# B&R Automation Studio project Nitto (part 7)

#### SPR_LabelerAut.st - Cam automat configuration for labeling unit
```iecst
(********************************************************************
 * COPYRIGHT -- Bernecker + Rainer
 ********************************************************************
 * Library: UserSpilke
 * File: SPR_LabelerAut.st
 * Author: knausenbergl
 * Created: January 30, 2013
 ********************************************************************
 * Implementation of library UserSpilke
 ********************************************************************)

(*<$Description$> Cam automat configuration for labeling unit </$Description$>*)
FUNCTION_BLOCK SPR_LabelerAut

	//********************	GLOBAL AUTOMAT CONFIGURATION ********************
	AutData.Master				:= Master;
	AutData.MaxMasterVelocity	:= MaxMasterVelocity;
	AutData.SlaveLatchParID		:= ACP10PAR_AUT_SL_S;
	AutData.StartState			:= 0;
	//***********************************************************************

	//********************	STATE 0: INIT ********************
	//state transition
	AutData.State[0].Event[0].Type		:= ncST_END;
	AutData.State[0].Event[0].Attribute	:= ncAT_ONCE;
	AutData.State[0].Event[0].NextState	:= 1;
	//********************************************************

	//********************	STATE 1: ALIGN MIDDLE OF CAM WITH REG MARK	********************
	//compensation
	AutData.State[1].CompMode	:= ncOFF;

	//cam profile
	AutData.State[1].CamProfileIndex	:= 16#FFFF;
//	AutData.State[1].MasterFactor		:= REAL_TO_UDINT(fmod( (LabelPeriod / 2.0 - DistanceToLabelSensor) , LabelPeriod) + 2.0 * LabelPeriod);
	AutData.State[1].MasterFactor		:= REAL_TO_UDINT(fmod( ABS(LabelPeriod / 2.0 - DistanceToLabelSensor) , LabelPeriod) + 2.0 * LabelPeriod);

	AutData.State[1].SlaveFactor		:= UDINT_TO_DINT(AutData.State[1].MasterFactor);

	//state transition
	AutData.State[1].Event[0].Type		:= ncST_END;
	AutData.State[1].Event[0].Attribute	:= ncAT_ONCE;
	AutData.State[1].Event[0].NextState	:= 2;
	//**************************************************************************************

	//********************	STATE 2: STANDARD CAM WITHOUT CORRECTION ********************
	//compensation
	AutData.State[2].CompMode			:= ncOFF;

	//cam profile
	AutData.State[2].CamProfileIndex	:= 16#FFFF;
	AutData.State[2].MasterFactor		:= REAL_TO_UDINT(LabelPeriod);
	AutData.State[2].SlaveFactor		:= REAL_TO_DINT(LabelPeriod);

	//state transition
	AutData.State[2].Event[0].Type		:= TriggerEvent;
	AutData.State[2].Event[0].Attribute	:= ncAT_ONCE;
	AutData.State[2].Event[0].NextState	:= 3;
	//************************************************************************

	//********************	STATE 3: LABEL POSITION CORRECTION	********************
	//compensation
	AutData.State[3].CompMode			:= ncSL_LATCHPOS;
	AutData.State[3].SlaveCompDistance	:= LabelPeriod;
	AutData.State[3].MasterCompDistance	:= LabelPeriod;

	//cam profile
	AutData.State[3].CamProfileIndex	:= 16#FFFE;
	AutData.State[3].MasterFactor		:= REAL_TO_UDINT(LabelPeriod);
	AutData.State[3].SlaveFactor		:= REAL_TO_DINT(LabelPeriod);

	//state transition
	AutData.State[3].Event[0].Type		:= TriggerEvent;
	AutData.State[3].Event[0].Attribute	:= ncAT_ONCE;
	AutData.State[3].Event[0].NextState	:= 3;

	AutData.State[3].Event[1].Type		:= ncST_END;
	AutData.State[3].Event[1].Attribute	:= ncAT_ONCE;
	AutData.State[3].Event[1].NextState	:= 4;
	//******************************************************************************

	//********************	STATE 4: POINT-TO-POINT CAM  WITHOUT CORRECTION	********************
	//compensation
	AutData.State[4].CompMode			:= ncWITH_CAM;
	AutData.State[4].SlaveCompDistance	:= LabelPeriod;
	AutData.State[4].MasterCompDistance	:= LabelPeriod;

	//cam profile
	AutData.State[4].CamProfileIndex	:= 16#FFFE;
	AutData.State[4].MasterFactor		:= REAL_TO_UDINT(LabelPeriod);
	AutData.State[4].SlaveFactor		:= REAL_TO_DINT(LabelPeriod);

	//state transition
	AutData.State[4].Event[0].Type		:= TriggerEvent;
	AutData.State[4].Event[0].Attribute	:= ncAT_ONCE;
	AutData.State[4].Event[0].NextState	:= 3;
	//*******************************************************************************************

	//ignore other states
	AutData.State[0].DisableStateInit	:= ncOFF;
	AutData.State[1].DisableStateInit	:= ncOFF;
	AutData.State[2].DisableStateInit	:= ncOFF;
	AutData.State[3].DisableStateInit	:= ncOFF;
	AutData.State[4].DisableStateInit	:= ncOFF;
	AutData.State[5].DisableStateInit	:= ncON;
	AutData.State[6].DisableStateInit	:= ncON;
	AutData.State[7].DisableStateInit	:= ncON;
	AutData.State[8].DisableStateInit	:= ncON;
	AutData.State[9].DisableStateInit	:= ncON;
	AutData.State[10].DisableStateInit	:= ncON;
	AutData.State[11].DisableStateInit	:= ncON;
	AutData.State[12].DisableStateInit	:= ncON;
	AutData.State[13].DisableStateInit	:= ncON;
	AutData.State[14].DisableStateInit	:= ncON;

	adrAutData	:= ADR(AutData);

END_FUNCTION_BLOCK
```

#### SPR_LabelerAutVax.st - Cam automat configuration for an "ideal" labeler (no label position correction)
```iecst
(********************************************************************
 * COPYRIGHT -- Bernecker + Rainer
 ********************************************************************
 * Library: UserSpilke
 * File: SPR_LabelerAutVax.st
 * Author: knausenbergl
 * Created: February 02, 2013
 ********************************************************************
 * Implementation of library UserSpilke
 ********************************************************************)

(*<$Description$> Cam automat configuration for an "ideal" labeler (no label position correction) </$Description$>*)
FUNCTION_BLOCK SPR_LabelerAutVax

	//the sum of acceleration distance, cam length and deceleration distance equals 1 label period
	IF ( (AccelerationBias >= 0.1) AND (AccelerationBias <= 10.0) ) THEN
		AccelerationDistance	:= (LabelPeriod - CamLength) * AccelerationBias / (AccelerationBias + 1.0);
	ELSE
		AccelerationDistance	:= (LabelPeriod - CamLength) / 2.0;	//default value
	END_IF;
	DecelerationDistance	:= LabelPeriod - CamLength - AccelerationDistance;

	//********************	GLOBAL AUTOMAT CONFIGURATION ********************
	AutData.Master				:= Master;
	AutData.MaxMasterVelocity	:= MaxMasterVelocity;
	AutData.StartState			:= 0;
	//***********************************************************************

	//********************	STATE 0: INIT ********************
	//state transition
	AutData.State[0].Event[0].Type		:= ncST_END;
	AutData.State[0].Event[0].Attribute	:= ncAT_ONCE;
	AutData.State[0].Event[0].NextState	:= 1;
	//********************************************************

	//********************	STATE 1: STANDSTILL, WAIT FOR TRIGGER EVENT	********************
	//compensation
	AutData.State[1].CompMode	:= ncOFF;

	//cam profile
	AutData.State[1].CamProfileIndex	:= 16#FFFF;
	AutData.State[1].MasterFactor		:= REAL_TO_UDINT(ProductLengthMaster);
	AutData.State[1].SlaveFactor		:= REAL_TO_DINT(LabelPeriod);

	//state transition
	AutData.State[1].Event[0].Type		:= ncSIGNAL1;
	AutData.State[1].Event[0].Attribute	:= ncAT_ONCE;
	AutData.State[1].Event[0].NextState	:= 2;

	AutData.State[1].Event[1].Type		:= TriggerEvent;	//reg mark found
	AutData.State[1].Event[1].Attribute	:= ncAT_ONCE;
	AutData.State[1].Event[1].NextState	:= 2;
	//**************************************************************************************

	//********************	STATE 2: DISPENSE FIRST LABEL ********************
	//compensation
//	AutData.State[2].CompMode			:= ncMA_LATCHPOS;
//	AutData.State[2].SlaveCompDistance	:= AccelerationDistance + 0.5 * CamLength;
//	AutData.State[2].MasterCompDistance	:= fmod( (DistanceToRmSensor - RegMarkPosition), ProductLengthMaster) + ProductLengthMaster;	//distance from sensor to middle of label

	// okrebs 12.09.13
	AutData.State[2].CompMode			:= ncMA_LATCHPOS;
	AutData.State[2].SlaveCompDistance	:= AccelerationDistance + 0.5 * LabelPeriod;
	AutData.State[2].MasterCompDistance	:= fmod( (DistanceToRmSensor - RegMarkPosition), ProductLengthMaster) + ProductLengthMaster;	//distance from sensor to middle of label

	//	//cam profile
    AutData.State[2].CamProfileIndex	:= 16#FFFF;
//	AutData.State[2].MasterFactor		:= REAL_TO_UDINT(CamLength);
//	AutData.State[2].SlaveFactor		:= REAL_TO_DINT(CamLength);

	IF (ProductLengthMaster > 0.0) THEN
		AutData.State[2].SlaveFactor		:= REAL_TO_DINT(LabelPeriod * LabelPeriod / ProductLengthMaster);
		AutData.State[2].MasterFactor		:= REAL_TO_UDINT(LabelPeriod);
	ELSE
		// Invalid parameters, use fix values
		AutData.State[2].MasterFactor		:= REAL_TO_UDINT(CamLength);
		AutData.State[2].SlaveFactor		:= REAL_TO_DINT(CamLength);
	END_IF

	//state transition
	AutData.State[2].Event[0].Type		:= ncST_END;
	AutData.State[2].Event[0].Attribute	:= ncAT_ONCE;
	AutData.State[2].Event[0].NextState	:= 3;

	AutData.State[2].Event[1].Type		:= ncSIGNAL2;	//stop labelling
	AutData.State[2].Event[1].Attribute	:= ncST_END;
	AutData.State[2].Event[1].NextState	:= 5;
	//************************************************************************

	//********************	STATE 3: CYCLIC LABELING WITHOUT CORRECTION	********************
	//compensation
	// AutData.State[3].CompMode			:= ncWITH_CAM;

	// okrebs 12.09.13
	 AutData.State[3].CompMode			:= ncOFF;

	AutData.State[3].SlaveCompDistance	:= LabelPeriod;			//label period on slave
	AutData.State[3].MasterCompDistance	:= ProductLengthMaster;	//distance label to label on master

//	//cam profile
//	AutData.State[3].CamProfileIndex	:= 16#FFFF;
//	AutData.State[3].MasterFactor		:= REAL_TO_UDINT(CamLength);
//	AutData.State[3].SlaveFactor		:= REAL_TO_DINT(CamLength);

	// okrebs / schoenefeldr 13.09.13
	AutData.State[3].CamProfileIndex	:= 16#FFFF;
	// Original:          SlaveFactor         Label period
	//            Gear = -------------- = -----------------------
	//                    MasterFactor      ProductLengthMaster
	// Use label period for the master cam length as it will be significantly
	// shorter than ProductLengthMaster -> so there is enough master distance
	// left for compensation:
	//           Label period                  Label period * (Label period / ProductLengthMaster)
	//   Gear = -----------------------  =   -------------------------
	//           ProductLengthMaster           Label period
	IF (ProductLengthMaster > 0.0) THEN
		AutData.State[3].SlaveFactor		:= REAL_TO_DINT(LabelPeriod * LabelPeriod / ProductLengthMaster);
		AutData.State[3].MasterFactor		:= REAL_TO_UDINT(LabelPeriod);
	ELSE
		// Invalid parameters, use fix values
		AutData.State[3].MasterFactor		:= REAL_TO_UDINT(CamLength);
		AutData.State[3].SlaveFactor		:= REAL_TO_DINT(CamLength);
	END_IF

	//state transition
	AutData.State[3].Event[0].Type		:= TriggerEvent;
	AutData.State[3].Event[0].Attribute	:= ncST_END;
	AutData.State[3].Event[0].NextState	:= 4;

	AutData.State[3].Event[1].Type		:= ncSIGNAL2;	//stop labelling
	AutData.State[3].Event[1].Attribute	:= ncST_END;
	AutData.State[3].Event[1].NextState	:= 5;

	//***************************************************************************************

	//********************	STATE 4: CYCLIC LABELING WITH CORRECTION	********************
	//compensation
	AutData.State[4].CompMode			:= ncMA_LATCHPOS;
	AutData.State[4].SlaveCompDistance	:= LabelPeriod;								//label period on slave
	AutData.State[4].MasterCompDistance	:= fmod( (DistanceToRmSensor - RegMarkPosition), ProductLengthMaster) + ProductLengthMaster;	//distance from sensor to middle of label

//	//cam profile
//	AutData.State[4].CamProfileIndex	:= 16#FFFF;
//	AutData.State[4].MasterFactor		:= REAL_TO_UDINT(CamLength);
//	AutData.State[4].SlaveFactor		:= REAL_TO_DINT(CamLength);

	// okrebs 12.09.13
	AutData.State[4].CamProfileIndex	:= 16#FFFF;
	AutData.State[4].MasterFactor		:= REAL_TO_UDINT(ProductLengthMaster);
	AutData.State[4].SlaveFactor		:= REAL_TO_DINT(LabelPeriod);

	IF (ProductLengthMaster > 0.0) THEN
		AutData.State[4].SlaveFactor		:= REAL_TO_DINT(LabelPeriod * LabelPeriod / ProductLengthMaster);
		AutData.State[4].MasterFactor		:= REAL_TO_UDINT(LabelPeriod);
	ELSE
		// Invalid parameters, use fix values
		AutData.State[4].MasterFactor		:= REAL_TO_UDINT(CamLength);
		AutData.State[4].SlaveFactor		:= REAL_TO_DINT(CamLength);
	END_IF

	//state transition
	AutData.State[4].Event[0].Type		:= TriggerEvent;
	AutData.State[4].Event[0].Attribute	:= ncST_END;
	AutData.State[4].Event[0].NextState	:= 4;

	AutData.State[4].Event[1].Type		:= ncSIGNAL2;	//stop labelling
	AutData.State[4].Event[1].Attribute	:= ncST_END;
	AutData.State[4].Event[1].NextState	:= 5;

	AutData.State[4].Event[2].Type		:= ncST_END;
	AutData.State[4].Event[2].Attribute	:= ncAT_ONCE;
	AutData.State[4].Event[2].NextState	:= 3;

	//***************************************************************************************

	//********************	STATE 5: DECELERATE TO STANDSTILL	********************
	//compensation
	AutData.State[5].CompMode			:= ncV_COMP_S_SL;
	AutData.State[5].SlaveCompDistance	:= DecelerationDistance;

	//cam profile
	AutData.State[5].CamProfileIndex	:= 16#FFFE;
	AutData.State[5].MasterFactor		:= REAL_TO_UDINT(CamLength);
	AutData.State[5].SlaveFactor		:= 0;

	//state transition
	AutData.State[5].Event[0].Type		:= ncST_END;
	AutData.State[5].Event[0].Attribute	:= ncAT_ONCE;
	AutData.State[5].Event[0].NextState	:= 1;
	//***************************************************************************************

	//ignore other states
	AutData.State[6].DisableStateInit	:= ncON;
	AutData.State[7].DisableStateInit	:= ncON;
	AutData.State[8].DisableStateInit	:= ncON;
	AutData.State[9].DisableStateInit	:= ncON;
	AutData.State[10].DisableStateInit	:= ncON;
	AutData.State[11].DisableStateInit	:= ncON;
	AutData.State[12].DisableStateInit	:= ncON;
	AutData.State[13].DisableStateInit	:= ncON;
	AutData.State[14].DisableStateInit	:= ncON;

	adrAutData	:= ADR(AutData);

END_FUNCTION_BLOCK
```

#### SPR_Punch.st - Implements the punch operation in automatic mode
```iecst
(********************************************************************
 * COPYRIGHT -- Bernecker + Rainer
 ********************************************************************
 * Library: UserSpilke
 * File: SPR_Punch.st
 * Author: knausenbergl
 * Created: November 09, 2012
 ********************************************************************
 * Implementation of library UserSpilke
 ********************************************************************)

(*<$Description$> Implements the punch operation in automatic mode </$Description$>*)
FUNCTION_BLOCK SPR_Punch

	IS.R_TRIG_Enable.CLK	:= Enable;
	IS.R_TRIG_Enable();

	IS.R_TRIG_Sync.CLK	:= Sync;
	IS.R_TRIG_Sync();

	EnableRestart	:= IS.EnableRestart;

	//experimental!!!!!!!!!!!!!!!!!!!!!!!
//	IF (Master <> 0) THEN
//		pMaster	ACCESS Master;
	//	END_IF;

	IS.MC_ReadActualPosition_0.Axis			:= Slave;
	IS.MC_ReadActualPosition_0.Enable		:= Enable;
	IS.MC_ReadActualPosition_0();

	IS.MC_ReadParameter_AxisPeriod.Axis				:= Slave;
	IS.MC_ReadParameter_AxisPeriod.ParameterNumber	:= 1008;	//axis modulo period
	IS.MC_ReadParameter_AxisPeriod.Enable			:= Enable;
	IS.MC_ReadParameter_AxisPeriod();
	//	IS.MC_BR_CrossCutterControl_0.AdvancedParameters.MasterStartDistance	:= DINT_TO_REAL(ProductLength);

	IF (IS.MC_ReadParameter_AxisPeriod.Value <> 0.0) THEN
		IS.NeutralPosition	:= fmod( (IS.MC_BR_CrossCutterControl_0.AdvancedParameters.CutPosition + IS.MC_ReadParameter_AxisPeriod.Value / 2.0), IS.MC_ReadParameter_AxisPeriod.Value);
//		IS.NeutralPosition	:= 0.0;			// Stanze ist nach Referenzfahrt in Position
	ELSE
		IS.NeutralPosition	:= 0.0;
	END_IF;

	//**********************	START OF STATE MACHINE	**************************
	//**********************	transitions from any state	**********************
	IF (NOT Enable) THEN
		Error		:= FALSE;
		ErrorID		:= 0;
		IS.State	:= SPR_STATE_DISABLED;
	ELSIF (IS.SPR_RmCapture_0.Error) THEN
		ErrorID		:= IS.SPR_RmCapture_0.ErrorID;
		Error		:= TRUE;
		IS.State	:= SPR_STATE_ERROR;
	ELSIF (IS.MC_BR_CrossCutterControl_0.Error) THEN
		ErrorID		:= IS.MC_BR_CrossCutterControl_0.ErrorID;
		Error		:= TRUE;
		IS.State	:= SPR_STATE_ERROR;
	ELSIF (IS.MC_BR_Phasing_0.Error) THEN
		ErrorID		:= IS.MC_BR_Phasing_0.ErrorID;
		Error		:= TRUE;
		IS.State	:= SPR_STATE_ERROR;
	ELSIF (IS.MC_BR_ReadAutPosition_0.Error) THEN
		ErrorID		:= IS.MC_BR_ReadAutPosition_0.ErrorID;
		Error		:= TRUE;
		IS.State	:= SPR_STATE_ERROR;
	ELSIF (IS.MC_MoveAbsolute_0.Error) THEN
		ErrorID		:= IS.MC_MoveAbsolute_0.ErrorID;
		Error		:= TRUE;
		IS.State	:= SPR_STATE_ERROR;
	ELSIF (IS.MC_ReadParameter_AxisPeriod.Error) THEN
		ErrorID		:= IS.MC_ReadParameter_AxisPeriod.ErrorID;
		Error		:= TRUE;
		IS.State	:= SPR_STATE_ERROR;
//	ELSIF (IS.MC_ReadParameter_MasterPeriod.Error) THEN
//		ErrorID		:= IS.MC_ReadParameter_MasterPeriod.ErrorID;
//		Error		:= TRUE;
//		IS.State	:= SPR_STATE_ERROR;
//	ELSIF (IS.MC_ReadActualPosition_Master.Error) THEN
//		ErrorID		:= IS.MC_ReadActualPosition_Master.ErrorID;
//		Error		:= TRUE;
//		IS.State	:= SPR_STATE_ERROR;
	END_IF;
	//****************************************************************************

	CASE (IS.State) OF
		//**********************	FUB inactive	**********************
		SPR_STATE_DISABLED:
			IS.MC_BR_ReadAutPosition_0.Execute		:= FALSE;
			IS.MC_MoveAbsolute_0.Execute			:= FALSE;
			IS.MC_BR_CrossCutterControl_0.Enable	:= FALSE;
			IS.MC_BR_CrossCutterControl_0.EnableCut	:= FALSE;
			IS.EnableRestart						:= FALSE;
			SetupComplete	:= FALSE;

			IF (Enable) THEN
				IS.State	:= SPR_STATE_INIT;
			END_IF;
		//****************************************************************

		//**********************	Internal variables are initialized	**********************
		SPR_STATE_INIT:
			IS.State	:= SPR_STATE_IDLE;
		//************************************************************************************

		//**********************	Waiting for a movement command	**********************
		SPR_STATE_IDLE:
			IF RestartAllowed THEN
				IS.EnableRestart						:= TRUE;
			END_IF;
			IF (EnableMove) THEN
				IS.MC_BR_CrossCutterControl_0.Enable	:= TRUE;
				IS.MC_BR_CrossCutterControl_0.EnableCut	:= FALSE;
				IS.State	:= SPR_STATE_CHECK_STANDBY;
			END_IF;
		//*********************************************************************************

		//**********************	Checking if automat restart is possible	**********************
		SPR_STATE_CHECK_STANDBY:
			IF (IS.MC_BR_CrossCutterControl_0.Active) THEN
				IS.MC_BR_CrossCutterControl_0.Enable	:= FALSE;
				IS.MC_BR_CrossCutterControl_0.EnableCut	:= FALSE;

				IF (IS.MC_BR_CrossCutterControl_0.StandBy AND IS.EnableRestart) THEN
					IS.MC_BR_ReadAutPosition_0.Execute		:= TRUE;
					IS.State	:= SPR_STATE_READ_AUT_POS;
				ELSE
					SetupComplete						:= FALSE;
					IS.MC_MoveAbsolute_0.Direction		:= mcPOSITIVE_DIR;
					IS.MC_MoveAbsolute_0.Position		:= IS.NeutralPosition;
					//					IS.MC_MoveAbsolute_0.Execute		:= TRUE;							// Keine Bewegung mehr auf die NeutralPosition
					// 2013-08-22 /scoenefeldr/
					IS.MC_BR_CrossCutterControl_0.AdvancedParameters.MasterStartDistance	:= IS.MC_BR_CrossCutterControl_0.AdvancedParameters.CutPosition - IS.MC_ReadActualPosition_0.Position;
					IF (IS.MC_BR_CrossCutterControl_0.AdvancedParameters.MasterStartDistance < 0) THEN
						IS.MC_BR_CrossCutterControl_0.AdvancedParameters.MasterStartDistance	:= IS.MC_BR_CrossCutterControl_0.AdvancedParameters.MasterStartDistance + ProductLength;
					ELSIF (IS.MC_BR_CrossCutterControl_0.AdvancedParameters.MasterStartDistance > ProductLength) THEN
						IS.MC_BR_CrossCutterControl_0.AdvancedParameters.MasterStartDistance	:= IS.MC_BR_CrossCutterControl_0.AdvancedParameters.MasterStartDistance - ProductLength;
					END_IF
					IS.State							:= SPR_STATE_MOVE_TO_NEUTRAL_POS;
				END_IF;
			END_IF;

			IF (NOT EnableMove) THEN
				IS.MC_BR_ReadAutPosition_0.Execute		:= FALSE;
				IS.MC_BR_CrossCutterControl_0.Enable	:= FALSE;
				IS.MC_BR_CrossCutterControl_0.EnableCut	:= FALSE;
				IS.State	:= SPR_STATE_IDLE;
			END_IF;
		//****************************************************************************************

		//**********************	Reading automat position	**********************
		SPR_STATE_READ_AUT_POS:
			IF (IS.MC_BR_ReadAutPosition_0.Done) THEN
				IS.MC_BR_ReadAutPosition_0.Execute	:= FALSE;
	//			IS.MC_MoveAbsolute_0.Direction		:= mcSHORTEST_WAY + mcAUTOMAT_POS;
				IS.MC_MoveAbsolute_0.Direction		:= mcPOSITIVE_DIR + mcAUTOMAT_POS;

				IS.MC_MoveAbsolute_0.Position		:= IS.MC_BR_ReadAutPosition_0.AutPosition;
				IS.MC_MoveAbsolute_0.Execute		:= TRUE;
				IS.State							:= SPR_STATE_MOVE_TO_AUT_POS;
			END_IF;

			IF (NOT EnableMove) THEN
				IS.MC_BR_ReadAutPosition_0.Execute	:= FALSE;
				IS.MC_MoveAbsolute_0.Execute		:= FALSE;
				IS.State	:= SPR_STATE_IDLE;
			END_IF;
		//*****************************************************************************

		//**********************	Moving to automat position	**********************
		SPR_STATE_MOVE_TO_AUT_POS:
			IF (IS.MC_MoveAbsolute_0.Done) THEN
				IS.MC_MoveAbsolute_0.Execute	:= FALSE;
				IS.MC_BR_CrossCutterControl_0.AdvancedParameters.StartMode	:= mcRESTART + mcCORRECT_CURRENT_CYCLE;
				IS.MC_BR_CrossCutterControl_0.Enable	:= TRUE;
				IS.MC_BR_CrossCutterControl_0.EnableCut	:= TRUE;
				IS.MC_BR_CrossCutterControl_0.AdvancedParameters.MasterMaxVelocity	:= AutPar.MaxMasterVelocity;
				IS.State	:= SPR_STATE_START_AUTOMAT;
			ELSIF (IS.MC_MoveAbsolute_0.CommandAborted) THEN
				IS.MC_MoveAbsolute_0.Execute	:= FALSE;
				IS.State	:= SPR_STATE_W4_RESET;
			END_IF;

			IF (NOT EnableMove) THEN
				IS.MC_MoveAbsolute_0.Execute			:= FALSE;
				IS.MC_BR_CrossCutterControl_0.Enable	:= FALSE;
				IS.MC_BR_CrossCutterControl_0.EnableCut	:= FALSE;
				IS.State	:= SPR_STATE_IDLE;
			END_IF;
		//*****************************************************************************

		//**********************	Moving to neutral position	**********************
		SPR_STATE_MOVE_TO_NEUTRAL_POS:
//			IF (IS.MC_MoveAbsolute_0.Done) THEN				//Keine Bewegung mehr auf die NeutralPosition
			IF (TRUE) THEN
				IS.MC_MoveAbsolute_0.Execute			:= FALSE;
				IS.MC_BR_CrossCutterControl_0.AdvancedParameters.StartMode	:=	mcIMMEDIATE + mcCORRECT_CURRENT_CYCLE;
				IS.MC_BR_CrossCutterControl_0.Enable	:= TRUE;
				IS.MC_BR_CrossCutterControl_0.EnableCut	:= TRUE;
				IS.MC_BR_CrossCutterControl_0.AdvancedParameters.MasterMaxVelocity	:= AutPar.StartMasterVelocity;
				IS.State	:= SPR_STATE_START_AUTOMAT;
				//experimental!!!!!!!!!!
//				IF (RegMarkPar.EnableRmCorrection) THEN
//					IS.MC_MoveAbsolute_0.Execute	:= FALSE;
//					IS.State						:= SPR_STATE_W4_REG_MARK;
//				ELSE
//					IS.MC_MoveAbsolute_0.Execute			:= FALSE;
//					IS.MC_BR_CrossCutterControl_0.AdvancedParameters.StartMode	:= mcIMMEDIATE + mcCORRECT_CURRENT_CYCLE;
//					IS.MC_BR_CrossCutterControl_0.Enable	:= TRUE;
//					IS.MC_BR_CrossCutterControl_0.EnableCut	:= TRUE;
//					IS.MC_BR_CrossCutterControl_0.AdvancedParameters.MasterMaxVelocity	:= AutPar.StartMasterVelocity;
//					IS.State	:= SPR_STATE_START_AUTOMAT;
//				END_IF;
			ELSIF (IS.MC_MoveAbsolute_0.CommandAborted) THEN
				IS.MC_MoveAbsolute_0.Execute	:= FALSE;
				IS.State	:= SPR_STATE_W4_RESET;
			END_IF;

			IF (NOT EnableMove) THEN
				IS.MC_MoveAbsolute_0.Execute			:= FALSE;
				IS.MC_BR_CrossCutterControl_0.Enable	:= FALSE;
				IS.MC_BR_CrossCutterControl_0.EnableCut	:= FALSE;
				IS.State	:= SPR_STATE_IDLE;
			END_IF;
		//*****************************************************************************

	//**********************	Starting cam automat	**********************
		SPR_STATE_START_AUTOMAT:
			IF (IS.MC_BR_CrossCutterControl_0.Active) THEN
				IS.EnableRestart	:= TRUE;
				IS.State			:= SPR_STATE_RUNNING;
			ELSIF (IS.MC_BR_CrossCutterControl_0.CommandAborted) THEN
				IS.MC_BR_CrossCutterControl_0.Enable	:= FALSE;
				IS.MC_BR_CrossCutterControl_0.EnableCut	:= FALSE;
				IS.State	:= SPR_STATE_W4_RESET;
			END_IF;

			IF (NOT EnableMove) THEN
				IS.MC_BR_CrossCutterControl_0.Enable	:= FALSE;
				IS.MC_BR_CrossCutterControl_0.EnableCut	:= FALSE;
				IS.State	:= SPR_STATE_IDLE;
			END_IF;
		//************************************************************************

		//**********************	Cam automat is running	**********************
		SPR_STATE_RUNNING:
			IF (IS.MC_BR_CrossCutterControl_0.CommandAborted) THEN
				IS.MC_BR_CrossCutterControl_0.Enable	:= FALSE;
				IS.MC_BR_CrossCutterControl_0.EnableCut	:= FALSE;
				IS.State	:= SPR_STATE_W4_RESET;
			END_IF;

			//cam automat synchronization movement is complete
			IF ( (IS.MC_BR_CrossCutterControl_0.IS.AutActStIdx >= 2) AND (IS.MC_BR_CrossCutterControl_0.IS.AutActStIdx <= 6) ) THEN
				SetupComplete	:= TRUE;
			END_IF;

			//set master speed to maximum velocity after start movement is complete
			IF (IS.MC_BR_CrossCutterControl_0.InCompensation) THEN
				IS.MC_BR_CrossCutterControl_0.AdvancedParameters.MasterMaxVelocity	:= AutPar.MaxMasterVelocity;
			END_IF;

			IF (NOT EnableMove) THEN
				IS.MC_BR_CrossCutterControl_0.Enable	:= FALSE;
				IS.MC_BR_CrossCutterControl_0.EnableCut	:= FALSE;
				IS.State	:= SPR_STATE_IDLE;
			END_IF;
		//************************************************************************

		//**********************	Command aborted, wait until "EnableMove" is reset	**********************
		SPR_STATE_W4_RESET:
			IF (NOT EnableMove) THEN
				IS.State	:= SPR_STATE_IDLE;
			END_IF;
		//************************************************************************

		//**********************	FUB Error	**********************
		SPR_STATE_ERROR:
		//************************************************************

		ELSE

	END_CASE;
	//**********************	END OF STATE MACHINE	************************

	//********************		Read automat position			********************
	IS.MC_BR_ReadAutPosition_0.Axis		:= Slave;
	IS.MC_BR_ReadAutPosition_0();
	//******************************************************************************

	//********************		Move absolute			********************
	IS.MC_MoveAbsolute_0.Axis			:= Slave;
	IS.MC_MoveAbsolute_0.Velocity		:= SetupPar.Velocity;
	IS.MC_MoveAbsolute_0.Acceleration	:= SetupPar.Acceleration;
	IS.MC_MoveAbsolute_0.Deceleration	:= SetupPar.Deceleration;
	IS.MC_MoveAbsolute_0();
	//**********************************************************************

	//********************		Reg mark detection			********************
	IS.SPR_RmCapture_0.Axis					:= RegMarkPar.Axis;
	IS.SPR_RmCapture_0.DistanceToSensor		:= RegMarkPar.DistanceToSensor;
	IS.SPR_RmCapture_0.ProductLength		:= ProductLength;
	IS.SPR_RmCapture_0.RegMarkPosition		:= RegMarkPar.RegMarkPosition;
	IS.SPR_RmCapture_0.TriggerInput			:= RegMarkPar.TriggerInput;
	IS.SPR_RmCapture_0.WindowNegative		:= RegMarkPar.WindowNegative;
	IS.SPR_RmCapture_0.WindowPositive		:= RegMarkPar.WindowPositive;

	IS.SPR_RmCapture_0.CutMasterPosition	:= IS.MC_BR_CrossCutterControl_0.CutMasterPosition - REAL_TO_DINT(IS.MC_BR_Phasing_0.Shift);
	IS.SPR_RmCapture_0.Enable				:= (IS.SPR_RmCapture_0.Enable OR Active) AND Enable AND RegMarkPar.EnableRmCorrection AND NOT RegMarkPar.EnableVRegMark;
	IS.SPR_RmCapture_0.SearchRM				:= SearchRM;
	IS.SPR_RmCapture_0();
	//**************************************************************************

	//*******************	Virtual Reg marks	********************
	IF RegMarkPar.EnableOffsetCorr THEN

		IS.SPR_RmCalcPosError_Virtual.RecordedValueValid	:= (IS.SPR_RmCalcPosError_Virtual.RecordedValue <> VRmRecordedPosition);
		IF (IS.MC_BR_CrossCutterControl_0.Active AND Enable AND RegMarkPar.EnableRmCorrection AND RegMarkPar.EnableVRegMark) THEN
			IF (IS.CutCount_1 > (IS.CutCntOld + 2)) AND NOT IS.OffsetErrorValid THEN
				IS.OffsetErrorValid		:= TRUE;
			END_IF
			IF IS.OffsetErrorValid THEN
				IF (IS.SPR_RmCalcPosError_Virtual.RecordedValue <> VRmRecordedPosition) THEN
					IS.OffsetValue := IS.OffsetValue + (VRmRecordedPosition - IS.SPR_RmCalcPosError_Virtual.RecordedValue) - ProductLength;
					IS.PositionError		:= RegMarkPar.RegMarkPosition - IS.OffsetValue;
	//				IS.PositionError		:= 0;
					IS.OffsetValue1		:= RegMarkPar.RegMarkPosition - IS.OffsetValue;
					IS.PositionErrorValid		:= TRUE;
				ELSE
					IS.PositionErrorValid		:= FALSE;
				END_IF
				IS.CutCntOld		:= IS.CutCount_1;
			ELSE
				IS.PositionError		:= 0;
			END_IF
		ELSE
	//		IS.OffsetValue := 0;
			IS.OffsetErrorValid := FALSE;
			IS.CutCntOld		:= IS.CutCount_1;
		END_IF

		IS.SPR_RmCalcPosError_Virtual.RecordedValue			:= VRmRecordedPosition;
		IS.SPR_RmCalcPosError_Virtual.CutMasterPosition		:= IS.MC_BR_CrossCutterControl_0.CutMasterPosition - REAL_TO_DINT(IS.MC_BR_Phasing_0.Shift);
	ELSE
		IS.SPR_RmCalcPosError_Virtual.Enable				:= (IS.SPR_RmCalcPosError_Virtual.Enable OR IS.MC_BR_CrossCutterControl_0.Active) AND Enable AND RegMarkPar.EnableRmCorrection AND RegMarkPar.EnableVRegMark;
		IS.SPR_RmCalcPosError_Virtual.DistanceToSensor		:= RegMarkPar.DistanceToSensor;
		IS.SPR_RmCalcPosError_Virtual.ProductLength			:= ProductLength;
		IS.SPR_RmCalcPosError_Virtual.RegMarkPosition		:= RegMarkPar.RegMarkPosition + VRmCorrection; // Änderung 05.06.13
		IS.SPR_RmCalcPosError_Virtual.RecordedValueValid	:= (IS.SPR_RmCalcPosError_Virtual.RecordedValue <> VRmRecordedPosition);
		IS.SPR_RmCalcPosError_Virtual.RecordedValue			:= VRmRecordedPosition;
		IS.SPR_RmCalcPosError_Virtual.CutMasterPosition		:= IS.MC_BR_CrossCutterControl_0.CutMasterPosition - REAL_TO_DINT(IS.MC_BR_Phasing_0.Shift);
		IS.SPR_RmCalcPosError_Virtual();

		IS.PositionError			:= IS.SPR_RmCalcPosError_Virtual.PositionError;
		IS.PositionErrorValid		:= IS.SPR_RmCalcPosError_Virtual.PositionErrorValid;

		IS.CutCntOld		:= IS.CutCount_1;
		IS.OffsetErrorValid		:= FALSE;
	END_IF
	//***************************************************************

	//limit correction value
	IS.LCRLimit_Correction.max_value	:= AutPar.MaxCorrection;
	IS.LCRLimit_Correction.min_value	:= - AutPar.MaxCorrection;

	//choose source of reg mark correction
	IF (RegMarkPar.EnableRmCorrection) THEN
		IF (RegMarkPar.EnableVRegMark) THEN
			IS.LCRLimit_Correction.in	:= IS.PositionError;
		ELSE
			IS.LCRLimit_Correction.in	:= IS.SPR_RmCapture_0.CorrectionValue;
		END_IF;
	ELSE
		IS.LCRLimit_Correction.in	:= 0.0;
	END_IF;
	IS.LCRLimit_Correction();

	//********************		CrossCutter			********************
	IS.MC_BR_CrossCutterControl_0.Master	:= Master;
	IS.MC_BR_CrossCutterControl_0.Slave		:= Slave;

	//calculate cut position within tool segment period
	IF (IS.MC_ReadParameter_AxisPeriod.Value <> 0.0) THEN
		IS.MC_BR_CrossCutterControl_0.CutRangeSlave		:= DINT_TO_REAL( (AutPar.CutEndPos - AutPar.CutStartPos) MOD REAL_TO_DINT(IS.MC_ReadParameter_AxisPeriod.Value) );
		IF (IS.MC_BR_CrossCutterControl_0.CutRangeSlave < 0.0) THEN
			IS.MC_BR_CrossCutterControl_0.CutRangeSlave	:= IS.MC_BR_CrossCutterControl_0.CutRangeSlave + IS.MC_ReadParameter_AxisPeriod.Value;
		END_IF;
		IS.MC_BR_CrossCutterControl_0.AdvancedParameters.CutPosition	:= DINT_TO_REAL( ( (AutPar.CutEndPos + AutPar.CutStartPos) / 2) MOD REAL_TO_DINT(IS.MC_ReadParameter_AxisPeriod.Value) );
		IF (IS.MC_BR_CrossCutterControl_0.AdvancedParameters.CutPosition < 0.0) THEN
			IS.MC_BR_CrossCutterControl_0.AdvancedParameters.CutPosition	:= IS.MC_BR_CrossCutterControl_0.AdvancedParameters.CutPosition + IS.MC_ReadParameter_AxisPeriod.Value;
		END_IF;

		//limit cut range of slave to avoid ACOPOS errors on wrong user input
		IF ( (AutPar.MinCutRangeSlave > 0.0) AND (AutPar.MinCutRangeSlave < IS.MC_ReadParameter_AxisPeriod.Value) ) THEN
			IS.MC_BR_CrossCutterControl_0.CutRangeSlave	:= MAX(IS.MC_BR_CrossCutterControl_0.CutRangeSlave, AutPar.MinCutRangeSlave);
		END_IF;
		IF ( (AutPar.MinCompRangeSlave > 0.0) AND (AutPar.MinCompRangeSlave < IS.MC_ReadParameter_AxisPeriod.Value) ) THEN
			IS.MC_BR_CrossCutterControl_0.CutRangeSlave := MIN(IS.MC_BR_CrossCutterControl_0.CutRangeSlave, (IS.MC_ReadParameter_AxisPeriod.Value - AutPar.MinCompRangeSlave) );
		END_IF;

		//scale cut range of master
		IS.LCRLimScal_CutRangeMaster.x1	:= 0.0;
		IS.LCRLimScal_CutRangeMaster.y1	:= IS.MC_BR_CrossCutterControl_0.CutRangeSlave;
		IS.LCRLimScal_CutRangeMaster.x2	:= 100.0;
		IS.LCRLimScal_CutRangeMaster.y2	:= (IS.MC_BR_CrossCutterControl_0.CutRangeSlave * ProductLength) / IS.MC_ReadParameter_AxisPeriod.Value;
		IS.LCRLimScal_CutRangeMaster.x	:= AutPar.Insetting;
		IS.LCRLimScal_CutRangeMaster();
		IS.MC_BR_CrossCutterControl_0.CutRangeMaster	:= IS.LCRLimScal_CutRangeMaster.y;
	ELSE
		IS.MC_BR_CrossCutterControl_0.CutRangeSlave						:= 0.0;
		IS.MC_BR_CrossCutterControl_0.CutRangeMaster					:= 0.0;
		IS.MC_BR_CrossCutterControl_0.AdvancedParameters.CutPosition	:= 0.0;
	END_IF;

	//init max. master velocity after start
	IS.R_TRIG_InCompensation.CLK	:= IS.MC_BR_CrossCutterControl_0.InCompensation;
	IS.R_TRIG_InCompensation();
	IS.CccInitMasterMaxVel	:= (IS.R_TRIG_InCompensation.Q AND (IS.MC_BR_CrossCutterControl_0.IS.AutActStIdx = 1) );

	IS.MC_BR_CrossCutterControl_0.ProductLength				:= ProductLength;
	IS.MC_BR_CrossCutterControl_0.ProductLengthCorrection	:= IS.LCRLimit_Correction.out;
	IS.MC_BR_CrossCutterControl_0.InitData					:=
	(IS.CccTriggerInit AND NOT RegMarkPar.EnableRmCorrection)
	OR IS.CccInitMasterMaxVel
	OR
	(
		RegMarkPar.EnableRmCorrection AND
		(
			(IS.SPR_RmCapture_0.CorrectionValid AND NOT RegMarkPar.EnableVRegMark)
//			OR (IS.SPR_RmCalcPosError_Virtual.PositionErrorValid AND RegMarkPar.EnableVRegMark)
			OR (IS.PositionErrorValid AND RegMarkPar.EnableVRegMark)
		)
	);

	IS.CutCount_1	:= IS.MC_BR_CrossCutterControl_0.CutCount;	 //save old value for change detection
	IS.MC_BR_CrossCutterControl_0();
	IS.CccTriggerInit	:= (IS.CutCount_1 <> IS.MC_BR_CrossCutterControl_0.CutCount);	//cut complete, trigger initialization
	//******************************************************************

	//********************	Phasing for synchronization movement	********************
	//TO DO: Shift value on the drive is not reset, even if phasing is disabled. ActualShiftValue may therefore lose resolution, as it is a REAL.
	IS.MC_BR_Phasing_0.Slave			:= Slave;
	IS.MC_BR_Phasing_0.Velocity			:= SyncPar.Velocity;
	IS.MC_BR_Phasing_0.Acceleration		:= SyncPar.Acceleration;
	IS.MC_BR_Phasing_0.ApplicationMode	:= mcTIME_BASED;
	IS.MC_BR_Phasing_0.ShiftMode		:= mcABSOLUTE_NO_RESET;

	IS.MC_BR_Phasing_0.Enable	:= (IS.MC_BR_Phasing_0.Enable OR IS.MC_BR_CrossCutterControl_0.Active) AND Enable;
	IS.MC_BR_Phasing_0.InitData	:= IS.R_TRIG_Sync.Q AND NOT IS.ShiftInProgress;

	IF (IS.MC_BR_Phasing_0.InitData) THEN
		IF (RegMarkPar.EnableVRegMark) THEN
			IF (RegMarkPar.EnableOffsetCorr) THEN
				IS.OffsetValue          := IS.OffsetValue + (VRmRecordedPosition - IS.SPR_RmCalcPosError_Virtual.RecordedValue) (*- ProductLength*);
				IS.PositionError        := RegMarkPar.RegMarkPosition - IS.OffsetValue;
				IS.RelativeShift        := - IS.PositionError MOD ProductLength;
				IS.OffsetValue			:= IS.OffsetValue - IS.RelativeShift;
				IS.PositionError		:= 0;  //PositionError wird durch MC_BR_Phasing korrigiert
			ELSE
				IS.RelativeShift        := - IS.SPR_RmCalcPosError_Virtual.PositionError MOD ProductLength;
			END_IF
		ELSE
			IS.RelativeShift        := - IS.SPR_RmCapture_0.CorrectionValue MOD ProductLength;
		END_IF;
		IF (IS.RelativeShift < 0) THEN
			IS.RelativeShift        := IS.RelativeShift + ProductLength;
		END_IF;
		IS.MC_BR_Phasing_0.Shift        := IS.MC_BR_Phasing_0.ActualShiftValue + DINT_TO_REAL(IS.RelativeShift);
	END_IF;

	IS.MC_BR_Phasing_0();

	//set a flag when a phase shift is in progress
	IF (IS.MC_BR_Phasing_0.ShiftAttained OR NOT IS.MC_BR_Phasing_0.Active) THEN
		IS.ShiftInProgress	:= FALSE;
	ELSIF (IS.MC_BR_Phasing_0.InitData) THEN
		IS.ShiftInProgress	:= TRUE;
	END_IF;
	//**********************************************************************************

	Active				:= IS.MC_BR_CrossCutterControl_0.Active (*OR (IS.State = SPR_STATE_W4_REG_MARK) OR (IS.State = SPR_STATE_START_AUTOMAT)*);
	CutMasterPosition	:= IS.MC_BR_CrossCutterControl_0.CutMasterPosition;

	//probe counter
	IF (Enable AND RegMarkPar.EnableRmCorrection) THEN
		IF (RegMarkPar.EnableVRegMark) THEN
			ProbeCounter		:= ProbeCounter + BOOL_TO_UDINT(IS.SPR_RmCalcPosError_Virtual.RecordedValueValid);
			MissedTriggers		:= 0;
			ActPositionError	:= IS.PositionError;
		ELSE
			ProbeCounter		:= IS.SPR_RmCapture_0.ProbeCounter;
			MissedTriggers		:= IS.SPR_RmCapture_0.MissedTriggers;
			ActPositionError	:= IS.SPR_RmCapture_0.CorrectionValue;
		END_IF;
	ELSE
		ProbeCounter		:= 0;
		MissedTriggers		:= 0;
		ActPositionError	:= 0;
	END_IF;

END_FUNCTION_BLOCK
```

#### FB_LaminateCTRL.st
```iecst
(********************************************************************
 * COPYRIGHT -- Microsoft
 ********************************************************************
 * Library: UserSpilke
 * Datei: FB_LaminateCTRL.st
 * Autor: Awalz
 * Erstellt: 9. Januar 2014
 ********************************************************************
 * Implementierung der Library UserSpilke
 ********************************************************************)

(* TODO: Bitte Kommentar hier einzufügen *)
FUNCTION_BLOCK FB_LaminateCTRL
	CASE StateCtrl OF
	(*	CTRL_FIRST_START:
			unitAxis.AxisStep := STATE_POWER_ON;
			unitAxis.MC_ReadStatus_0.Enable := TRUE;
		(*	IF (NOT Enable) THEN
				Error		:= FALSE;
				ErrorID		:= 0;
				IS.State	:= SPR_STATE_DISABLED;
			ELSIF (IS.SPR_RmCapture_0.Error) THEN
				ErrorID		:= IS.SPR_RmCapture_0.ErrorID;
				Error		:= TRUE;
				IS.State	:= SPR_STATE_ERROR;
			ELSIF (IS.MC_BR_CrossCutterControl_0.Error) THEN
				ErrorID		:= IS.MC_BR_CrossCutterControl_0.ErrorID;
				Error		:= TRUE;
				IS.State	:= SPR_STATE_ERROR;
			ELSIF (IS.MC_BR_Phasing_0.Error) THEN
				ErrorID		:= IS.MC_BR_Phasing_0.ErrorID;
				Error		:= TRUE;
				IS.State	:= SPR_STATE_ERROR;
			ELSIF (IS.MC_BR_ReadAutPosition_0.Error) THEN
				ErrorID		:= IS.MC_BR_ReadAutPosition_0.ErrorID;
				Error		:= TRUE;
				IS.State	:= SPR_STATE_ERROR;
			ELSIF (IS.MC_MoveAbsolute_0.Error) THEN
				ErrorID		:= IS.MC_MoveAbsolute_0.ErrorID;
				Error		:= TRUE;
				IS.State	:= SPR_STATE_ERROR;
			ELSIF (IS.MC_ReadParameter_AxisPeriod.Error) THEN
				ErrorID		:= IS.MC_ReadParameter_AxisPeriod.ErrorID;
				Error		:= TRUE;
				IS.State	:= SPR_STATE_ERROR;
		(*	status := unitAxis.MC_ReadStatus_0.ErrorID ;*)

	(*	CTRL_MANUAL_BEFORE: ;
		(*unitAxis.BasicControl.*)

	(*	CTRL_MANUAL: ;
			unitAxis.MC_GearIn_0.Execute := TRUE;
			unitAxis.MC_GearIn_0.Master := machineMaster;
			(*unitAxis.MC_GearIn_0.Slave :=
			(*IF unitAxis.MC_ReadAxisError_0 = AxisCMD
		CTRL_MANUAL_BEFORE:
			unitAxis.AxisStep := AxisCMD

		(*	unitAxis.Axis1Obj 	:=
			(*cutterAxis.drvCtrl.ncError(InstanceId := status.id, StationName := status.name, ErrorId := CONST.CUTTINGUNIT.ERRORS.AXISERROR);
			cutterAxis.drvCtrl.safetySpeedMessage(InstanceId := status.id, StationName := status.name, ErrorId := CONST.CUTTINGUNIT.ERRORS.SAFETY_SPEED);
			schutzhauben.vorn.err(InstanceId := status.id, StationName := status.name, ErrorId := CONST.CUTTINGUNIT.ERRORS.HAUBE1_VORN_OFFEN );
			schutzhauben.hinten.err(InstanceId := status.id, StationName := status.name, ErrorId := CONST.CUTTINGUNIT.ERRORS.HAUBE2_HINTEN_OFFEN );
			data.tool.calcPerimeters();

			status.Init(recipeMode := data.recipe.mode);
			busy := TRUE;
			StateCtrl := CTRL_EMERGENCYSTOP_BEFORE;*)

	END_CASE

END_FUNCTION_BLOCK
```

#### FB_AxisCtlr.st
```iecst
(********************************************************************
 * COPYRIGHT -- Microsoft
 ********************************************************************
 * Library: UserSpilke
 * Datei: FB_AxisCtlr.st
 * Autor: Awalz
 * Erstellt: 12. Januar 2014
 ********************************************************************
 * Implementierung der Library UserSpilke
 ********************************************************************)

(* TODO: Bitte Kommentar hier einzufügen *)
(*FUNCTION_BLOCK FB_AxisCtrl
(***************************************************************
        Control Sequence
***************************************************************)
(* status information is read before the step sequencer to attain a shorter reaction time *)
(************************ MC_READSTATUS *************************)
//	MC_ReadStatus_0.Enable := NOT(MC_ReadStatus_0.Error);
//	MC_ReadStatus_0.Axis := Axis1Obj;
//	MC_ReadStatus_0();
//	BasicControl.AxisState.Disabled             := MC_ReadStatus_0.Disabled;
//	BasicControl.AxisState.StandStill           := MC_ReadStatus_0.StandStill;
//	BasicControl.AxisState.Stopping             := MC_ReadStatus_0.Stopping;
//	BasicControl.AxisState.Homing               := MC_ReadStatus_0.Homing;
//	BasicControl.AxisState.DiscreteMotion       := MC_ReadStatus_0.DiscreteMotion;
//	BasicControl.AxisState.ContinuousMotion     := MC_ReadStatus_0.ContinuousMotion;
//	BasicControl.AxisState.SynchronizedMotion   := MC_ReadStatus_0.SynchronizedMotion;
//	BasicControl.AxisState.ErrorStop            := MC_ReadStatus_0.Errorstop;
//
//	(********************MC_BR_READDRIVESTATUS***********************)
//	MC_BR_ReadDriveStatus_0.Enable := NOT(MC_BR_ReadDriveStatus_0.Error);
//	MC_BR_ReadDriveStatus_0.Axis := Axis1Obj;
//	MC_BR_ReadDriveStatus_0.AdrDriveStatus := ADR(BasicControl.Status.DriveStatus);
//	MC_BR_ReadDriveStatus_0();
//
//	(******************** MC_READACTUALPOSITION *********************)
//	MC_ReadActualPosition_0.Enable := (NOT(MC_ReadActualPosition_0.Error));
//	MC_ReadActualPosition_0.Axis := Axis1Obj;
//	MC_ReadActualPosition_0();
//	IF(MC_ReadActualPosition_0.Valid = TRUE)THEN
//		BasicControl.Status.ActPosition := MC_ReadActualPosition_0.Position;
//	END_IF
//
//	(******************** MC_READACTUALVELOCITY *********************)
//	MC_ReadActualVelocity_0.Enable := (NOT(MC_ReadActualVelocity_0.Error));
//	MC_ReadActualVelocity_0.Axis := Axis1Obj;
//	MC_ReadActualVelocity_0();
//	IF(MC_ReadActualVelocity_0.Valid = TRUE)THEN
//		BasicControl.Status.ActVelocity := MC_ReadActualVelocity_0.Velocity;
//	END_IF
//
//	(************************ MC_READAXISERROR **********************)
//	MC_ReadAxisError_0.Enable := NOT(MC_ReadAxisError_0.Error);
//	MC_ReadAxisError_0.Axis := Axis1Obj;
//	MC_ReadAxisError_0.DataAddress := ADR(BasicControl.Status.ErrorText);
//	MC_ReadAxisError_0.DataLength := SIZEOF(BasicControl.Status.ErrorText);
//	MC_ReadAxisError_0.DataObjectName := 'acp10etxen';
//	MC_ReadAxisError_0();
//
//	(* central monitoring OF stop command attains a shorter reaction TIME in CASE OF emergency stop *)
//	(******************CHECK FOR STOP COMMAND************************)
//	IF (BasicControl.Command.Stop = TRUE) THEN
//		IF ((AxisStep >= STATE_READY) AND (AxisStep < STATE_ERROR)) THEN
//			(* reset all FB execute inputs we use *)
//			MC_Home_0.Execute := 0;
//			MC_Stop_0.Execute := 0;
//			MC_MoveAbsolute_0.Execute := 0;
//			MC_MoveAdditive_0.Execute := 0;
//			MC_MoveVelocity_0.Execute := 0;
//			MC_ReadAxisError_0.Acknowledge := 0;
//			MC_Reset_0.Execute := 0;
//
//			(* reset user commands *)
//			BasicControl.Command.Stop := 0;
//			BasicControl.Command.Home := 0;
//			BasicControl.Command.MoveJogPos := 0;
//			BasicControl.Command.MoveJogNeg := 0;
//			BasicControl.Command.MoveVelocity := 0;
//			BasicControl.Command.MoveAbsolute := 0;
//			BasicControl.Command.MoveAdditive := 0;
//			AxisStep := STATE_STOP;
//		END_IF
//	END_IF
//
//	(**************** CHECK FOR GENERAL AXIS ERROR ******************)
//	IF ((MC_ReadAxisError_0.AxisErrorID <> 0) AND (MC_ReadAxisError_0.Valid = TRUE)) THEN
//		AxisStep := STATE_ERROR_AXIS;
//		(***************** CHECK IF POWER SHOULD BE OFF *******************)
//	ELSIF ((BasicControl.Command.Power = FALSE) AND (MC_ReadAxisError_0.Valid = TRUE)) THEN
//		IF ((MC_ReadStatus_0.Errorstop = TRUE) AND (MC_ReadStatus_0.Valid = TRUE)) THEN
//			AxisStep := STATE_ERROR_RESET;
//		ELSE
//			AxisStep := STATE_WAIT;
//		END_IF
//	END_IF
//
//	CASE AxisStep OF
//
//		(******************** WAIT *************************)
//		STATE_WAIT:  (* STATE: Wait *)
//			IF (BasicControl.Command.Power = TRUE) THEN
//				AxisStep := STATE_POWER_ON;
//			ELSE
//				MC_Power_0.Enable := FALSE;
//			END_IF
//
//			(* reset all FB execute inputs we use *)
//			MC_Home_0.Execute := FALSE;
//			MC_Stop_0.Execute := FALSE;
//			MC_MoveAbsolute_0.Execute := FALSE;
//			MC_MoveAdditive_0.Execute := FALSE;
//			MC_MoveVelocity_0.Execute := FALSE;
//			MC_ReadAxisError_0.Acknowledge := FALSE;
//			MC_Reset_0.Execute := FALSE;
//
//			(* reset user commands *)
//			BasicControl.Command.Stop := FALSE;
//			BasicControl.Command.Home := FALSE;
//			BasicControl.Command.MoveJogPos := FALSE;
//			BasicControl.Command.MoveJogNeg := FALSE;
//			BasicControl.Command.MoveVelocity := FALSE;
//			BasicControl.Command.MoveAbsolute := FALSE;
//			BasicControl.Command.MoveAdditive := FALSE;
//
//			BasicControl.Status.ErrorID := 0;
//
//		(******************** POWER ON **********************)
//		STATE_POWER_ON:  (* STATE: Power on *)
//			MC_Power_0.Enable := TRUE;
//			IF (MC_Power_0.Status = TRUE) THEN
//				AxisStep := STATE_READY;
//			END_IF
//			(* if a power error occured go to error state *)
//			IF (MC_Power_0.Error = TRUE) THEN
//				BasicControl.Status.ErrorID := MC_Power_0.ErrorID;
//				AxisStep := STATE_ERROR;
//			END_IF
//
//		(******************** READY **********************)
//		STATE_READY:  (* STATE: Waiting for commands *)
//			IF (BasicControl.Command.Home = TRUE)THEN
//				BasicControl.Command.Home := FALSE;
//				AxisStep := STATE_HOME;
//
//			ELSIF (BasicControl.Command.Stop = TRUE) THEN
//				AxisStep := STATE_STOP;
//
//			ELSIF (BasicControl.Command.MoveJogPos = TRUE) THEN
//				AxisStep := STATE_JOG_POSITIVE;
//
//			ELSIF (BasicControl.Command.MoveJogNeg = TRUE) THEN
//				AxisStep := STATE_JOG_NEGATIVE;
//
//			ELSIF (BasicControl.Command.MoveAbsolute = TRUE) THEN
//				BasicControl.Command.MoveAbsolute := FALSE;
//				AxisStep := STATE_MOVE_ABSOLUTE;
//
//			ELSIF (BasicControl.Command.MoveAdditive = TRUE) THEN
//				BasicControl.Command.MoveAdditive := FALSE;
//				AxisStep := STATE_MOVE_ADDITIVE;
//
//			ELSIF (BasicControl.Command.MoveVelocity = TRUE) THEN
//				BasicControl.Command.MoveVelocity := FALSE;
//				AxisStep := STATE_MOVE_VELOCITY;
//
//			ELSIF (BasicControl.Command.Halt = TRUE) THEN
//				BasicControl.Command.Halt := FALSE;
//				AxisStep := STATE_HALT;
//			END_IF
//
//		(******************** HOME **********************)
//		STATE_HOME:  (* STATE: start homing process *)
//			MC_Home_0.Position := BasicControl.Parameter.HomePosition;
//			MC_Home_0.HomingMode := BasicControl.Parameter.HomeMode;
//			MC_Home_0.Execute := TRUE;
//			IF (MC_Home_0.Done = TRUE) THEN
//				MC_Home_0.Execute := FALSE;
//				AxisStep := STATE_READY;
//			END_IF
//			(* if a homing error occured go to error state *)
//			IF (MC_Home_0.Error = TRUE) THEN
//				MC_Home_0.Execute := FALSE;
//				BasicControl.Status.ErrorID := MC_Home_0.ErrorID;
//				AxisStep := STATE_ERROR;
//			END_IF
//
//		(***********************HALT_MOVEMENT***************************)
//		STATE_HALT:   (* STATE: Halt movement *)
//			MC_Halt_0.Deceleration := BasicControl.Parameter.Deceleration;
//			MC_Halt_0.Execute := TRUE;
//			IF (MC_Halt_0.Done = TRUE) THEN
//				MC_Halt_0.Execute := FALSE;
//				AxisStep := STATE_READY;
//			END_IF
//			(* check if error occured *)
//			IF (MC_Halt_0.Error = TRUE) THEN
//				BasicControl.Status.ErrorID := MC_Halt_0.ErrorID;
//				MC_Halt_0.Execute := FALSE;
//				AxisStep := STATE_ERROR;
//			END_IF
//
//		(*********************** STOP MOVEMENT *************************)
//		STATE_STOP:  (* STATE: Stop movement *)
//			MC_Stop_0.Deceleration := BasicControl.Parameter.Deceleration;
//			MC_Stop_0.Execute := TRUE;
//			(* if axis is stopped go to ready state *)
//			IF ((MC_Stop_0.Done = TRUE) AND (BasicControl.Command.Stop = FALSE)) THEN
//				MC_Stop_0.Execute := FALSE;
//				AxisStep := STATE_READY;
//			END_IF
//			(* check if error occured *)
//			IF (MC_Stop_0.Error = TRUE) THEN
//				BasicControl.Status.ErrorID := MC_Stop_0.ErrorID;
//				MC_Stop_0.Execute := FALSE;
//				AxisStep := STATE_ERROR;
//			END_IF
//
//		(******************** START JOG MOVEMENT POSITVE **********************)
//		STATE_JOG_POSITIVE:  (* STATE: Start jog movement in positive direction *)
//			MC_MoveVelocity_0.Velocity      := BasicControl.Parameter.JogVelocity;
//			MC_MoveVelocity_0.Acceleration  := BasicControl.Parameter.Acceleration;
//			MC_MoveVelocity_0.Deceleration  := BasicControl.Parameter.Deceleration;
//			MC_MoveVelocity_0.Direction     := mcPOSITIVE_DIR;
//			MC_MoveVelocity_0.Execute := TRUE;
//			IF (BasicControl.Command.MoveJogPos = FALSE) THEN
//				MC_MoveVelocity_0.Execute := FALSE;
//				AxisStep := STATE_HALT;
//			END_IF
//			(* check if error occured *)
//			IF (MC_MoveVelocity_0.Error = TRUE) THEN
//				BasicControl.Status.ErrorID := MC_MoveVelocity_0.ErrorID;
//				MC_MoveVelocity_0.Execute := FALSE;
//				AxisStep := STATE_ERROR;
//			END_IF
//
//		(******************** START JOG MOVEMENT NEGATIVE **********************)
//		STATE_JOG_NEGATIVE:  (* STATE: Start jog movement in negative direction *)
//			MC_MoveVelocity_0.Velocity      := BasicControl.Parameter.JogVelocity;
//			MC_MoveVelocity_0.Acceleration  := BasicControl.Parameter.Acceleration;
//			MC_MoveVelocity_0.Deceleration  := BasicControl.Parameter.Deceleration;
//			MC_MoveVelocity_0.Direction	    := mcNEGATIVE_DIR;
//			MC_MoveVelocity_0.Execute := TRUE;
//			IF (BasicControl.Command.MoveJogNeg = FALSE) THEN
//				MC_MoveVelocity_0.Execute := FALSE;
//				AxisStep := STATE_HALT;
//			END_IF
//			(* check if error occured *)
//			IF (MC_MoveVelocity_0.Error = TRUE) THEN
//				BasicControl.Status.ErrorID := MC_MoveVelocity_0.ErrorID;
//				MC_MoveVelocity_0.Execute := FALSE;
//				AxisStep := STATE_ERROR;
//			END_IF
//
//		(******************** START ABSOLUTE MOVEMENT **********************)
//		STATE_MOVE_ABSOLUTE:  (* STATE: Start absolute movement *)
//			MC_MoveAbsolute_0.Position      := BasicControl.Parameter.Position;
//			MC_MoveAbsolute_0.Velocity      := BasicControl.Parameter.Velocity;
//			MC_MoveAbsolute_0.Acceleration  := BasicControl.Parameter.Acceleration;
//			MC_MoveAbsolute_0.Deceleration  := BasicControl.Parameter.Deceleration;
//			MC_MoveAbsolute_0.Direction     := BasicControl.Parameter.Direction;
//			MC_MoveAbsolute_0.Execute := TRUE;
//			(* check if commanded position is reached *)
//			IF (BasicControl.Command.Halt) THEN
//				BasicControl.Command.Halt := FALSE;
//				MC_MoveAbsolute_0.Execute := FALSE;
//				AxisStep := STATE_HALT;
//			ELSIF (MC_MoveAbsolute_0.Done = TRUE) THEN
//				MC_MoveAbsolute_0.Execute := FALSE;
//				AxisStep := STATE_READY;
//			END_IF
//			(* check if error occured *)
//			IF (MC_MoveAbsolute_0.Error = TRUE) THEN
//				BasicControl.Status.ErrorID := MC_MoveAbsolute_0.ErrorID;
//				MC_MoveAbsolute_0.Execute := TRUE;
//				AxisStep := STATE_ERROR;
//			END_IF
//
//		(******************** START ADDITIVE MOVEMENT **********************)
//		STATE_MOVE_ADDITIVE:  (* STATE: Start additive movement *)
//			MC_MoveAdditive_0.Distance      := BasicControl.Parameter.Distance;
//			MC_MoveAdditive_0.Velocity      := BasicControl.Parameter.Velocity;
//			MC_MoveAdditive_0.Acceleration  := BasicControl.Parameter.Acceleration;
//			MC_MoveAdditive_0.Deceleration  := BasicControl.Parameter.Deceleration;
//			MC_MoveAdditive_0.Execute := TRUE;
//			(* check if commanded distance is reached *)
//			IF (BasicControl.Command.Halt) THEN
//				BasicControl.Command.Halt := FALSE;
//				MC_MoveAdditive_0.Execute := FALSE;
//				AxisStep := STATE_HALT;
//			ELSIF (MC_MoveAdditive_0.Done = TRUE) THEN
//				MC_MoveAdditive_0.Execute := FALSE;
//				AxisStep := STATE_READY;
//			END_IF
//			(* check if error occured *)
//			IF (MC_MoveAdditive_0.Error = TRUE) THEN
//				BasicControl.Status.ErrorID := MC_MoveAdditive_0.ErrorID;
//				MC_MoveAdditive_0.Execute := FALSE;
//				AxisStep := STATE_ERROR;
//			END_IF
//
//		(******************** START VELOCITY MOVEMENT **********************)
//		STATE_MOVE_VELOCITY:  (* STATE: Start velocity movement *)
//			MC_MoveVelocity_0.Velocity      := BasicControl.Parameter.Velocity;
//			MC_MoveVelocity_0.Acceleration  := BasicControl.Parameter.Acceleration;
//			MC_MoveVelocity_0.Deceleration  := BasicControl.Parameter.Deceleration;
//			MC_MoveVelocity_0.Direction     := BasicControl.Parameter.Direction;
//			MC_MoveVelocity_0.Execute := TRUE;
//			(* check if commanded velocity is reached *)
//			IF (BasicControl.Command.Halt) THEN
//				BasicControl.Command.Halt := FALSE;
//				MC_MoveVelocity_0.Execute := FALSE;
//				AxisStep := STATE_HALT;
//			ELSIF (MC_MoveVelocity_0.InVelocity = TRUE) THEN
//				MC_MoveVelocity_0.Execute := FALSE;
//				AxisStep := STATE_READY;
//			END_IF
//			(* check if error occured *)
//			IF (MC_MoveVelocity_0.Error = TRUE) THEN
//				BasicControl.Status.ErrorID := MC_MoveVelocity_0.ErrorID;
//				MC_MoveVelocity_0.Execute := FALSE;
//				AxisStep := STATE_ERROR;
//			END_IF
//
//		(******************** FB-ERROR OCCURED *************************)
//		STATE_ERROR:  (* STATE: Error *)
//			(* check if FB indicates an axis error *)
//			IF (MC_ReadAxisError_0.AxisErrorCount<>0) THEN
//				AxisStep := STATE_ERROR_AXIS;
//			ELSE
//				IF (BasicControl.Command.ErrorAcknowledge = TRUE) THEN
//					BasicControl.Command.ErrorAcknowledge := FALSE;
//					BasicControl.Status.ErrorID := 0;
//					(* reset axis if it is in axis state ErrorStop *)
//					IF ((MC_ReadStatus_0.Errorstop = TRUE) AND (MC_ReadStatus_0.Valid = TRUE)) THEN
//						AxisStep := STATE_ERROR_RESET;
//					ELSE
//						AxisStep := STATE_WAIT;
//					END_IF
//				END_IF
//			END_IF
//
//		(******************** AXIS-ERROR OCCURED *************************)
//		STATE_ERROR_AXIS:  (* STATE: Axis Error *)
//			IF (MC_ReadAxisError_0.Valid = TRUE) THEN
//				IF (MC_ReadAxisError_0.AxisErrorID <> 0) THEN
//					BasicControl.Status.ErrorID := MC_ReadAxisError_0.AxisErrorID;
//				END_IF
//				MC_ReadAxisError_0.Acknowledge := FALSE;
//				IF (BasicControl.Command.ErrorAcknowledge = TRUE) THEN
//					BasicControl.Command.ErrorAcknowledge := FALSE;
//					(* acknowledge axis error *)
//					IF (MC_ReadAxisError_0.AxisErrorID <> 0) THEN
//						MC_ReadAxisError_0.Acknowledge := TRUE;
//					END_IF
//				END_IF
//				IF (MC_ReadAxisError_0.AxisErrorCount = 0) THEN
//					(* reset axis if it is in axis state ErrorStop *)
//					BasicControl.Status.ErrorID := 0;
//					IF ((MC_ReadStatus_0.Errorstop = TRUE) AND (MC_ReadStatus_0.Valid = TRUE)) THEN
//						AxisStep := STATE_ERROR_RESET;
//					ELSE
//						AxisStep := STATE_WAIT;
//					END_IF
//				END_IF
//			END_IF
//
//		(******************** RESET DONE *************************)
//		STATE_ERROR_RESET:  (* STATE: Wait for reset done *)
//			MC_Reset_0.Execute := TRUE;
//			(* reset MC_Power.Enable if this FB is in Error*)
//			IF (MC_Power_0.Error = TRUE) THEN
//				MC_Power_0.Enable := FALSE;
//			END_IF
//			IF(MC_Reset_0.Done = TRUE)THEN
//				MC_Reset_0.Execute := FALSE;
//				AxisStep := STATE_WAIT;
//			ELSIF(MC_Reset_0.Error = TRUE) THEN
//				MC_Reset_0.Execute := FALSE;
//				AxisStep := STATE_ERROR;
//			END_IF
//			(******************** SEQUENCE END *************************)
//	END_CASE
//
//(***************************************************************
//        Function Block Calls
//***************************************************************)
//
//(************************** MC_POWER ****************************)
//	MC_Power_0.Axis := Axis1Obj;  (* pointer to axis *)
//	MC_Power_0();
//
//	(************************** MC_HOME *****************************)
//	MC_Home_0.Axis := Axis1Obj;
//	MC_Home_0();
//
//	(********************** MC_MOVEABSOLUTE *************************)
//	MC_MoveAbsolute_0.Axis := Axis1Obj;
//	MC_MoveAbsolute_0();
//
//	(********************** MC_MOVEADDITIVE *************************)
//	MC_MoveAdditive_0.Axis := Axis1Obj;
//	MC_MoveAdditive_0();
//
//	(********************** MC_MOVEVELOCITY *************************)
//	MC_MoveVelocity_0.Axis := Axis1Obj;
//	MC_MoveVelocity_0();
//
//	(************************** MC_STOP *****************************)
//	MC_Stop_0.Axis := Axis1Obj;
//	MC_Stop_0();
//
//	(***************************MC_HALT******************************)
//	MC_Halt_0.Axis := Axis1Obj;
//	MC_Halt_0();
//
//	(************************** MC_RESET ****************************)
//	MC_Reset_0.Axis := Axis1Obj;
//	MC_Reset_0();
(*END_FUNCTION_BLOCK*)
```

#### FB_MainCtrl.st
```iecst
(********************************************************************
 * COPYRIGHT -- Microsoft
 ********************************************************************
 * Library: UserSpilke
 * Datei: FB_MainCtrl.st
 * Autor: Awalz
 * Erstellt: 24. März 2014
 ********************************************************************
 * Implementierung der Library UserSpilke
 ********************************************************************)

(* TODO: Daten FB dient als Datenstruktur *)
FUNCTION_BLOCK FB_MainCtrl
END_FUNCTION_BLOCK
```

#### FB_MainHW.st
```iecst
(********************************************************************
 * COPYRIGHT -- Microsoft
 ********************************************************************
 * Library: UserSpilke
 * Datei: FB_MainHW.st
 * Autor: Awalz
 * Erstellt: 26. März 2014
 ********************************************************************
 * Implementierung der Library UserSpilke
 ********************************************************************)

(*<$Description$> TODO: Bitte Kommentar hier einzufügen </$Description$>*)
FUNCTION_BLOCK FB_MainHW
END_FUNCTION_BLOCK
```

### Library Logical/Libraries/SprMachine (IEC, version 1.00.0) - Control and monitoring of the whole machine

#### SprMachine.typ - Exported data types
```iecst
(********************************************************************
 * COPYRIGHT -- Bernecker + Rainer
 ********************************************************************
 * Library: SprMachine
 * File: SprMachine.typ
 * Author: knausenbergl
 * Created: December 21, 2012
 ********************************************************************
 * Data types of library SprMachine
 ********************************************************************)

TYPE
	emuSprMachine_PowerState :
		(
		SPR_MACH_PWR_DISABLED,
		SPR_MACH_PWR_ENABLED,
		SPR_MACH_PWR_ESTOP_AUTO,
		SPR_MACH_PWR_DELAY_24V_OFF,
		SPR_MACH_PWR_ERROR
		);
END_TYPE
```

#### SprMachine.fun - Exported functions and function blocks
```iecst
(********************************************************************
 * COPYRIGHT -- Bernecker + Rainer
 ********************************************************************
 * Library: SprMachine
 * File: SprMachine.fun
 * Author: knausenbergl
 * Created: December 21, 2012
 ********************************************************************
 * Functions and function blocks of library SprMachine
 ********************************************************************)

FUNCTION_BLOCK SPR_MachinePower (*Power on/off drives*)
	VAR_INPUT
		SwitchOn : BOOL; (*Command to switch on power*)
		SwitchOff : BOOL; (*Command to switch off power*)
		SafetyOk : BOOL; (*Safety OK, no EStop requested*)
		SwitchOffDelay : TIME; (*Delay for switching off 24V control voltage e.g. in the case of an EStop*)
		AutoModeActive : BOOL; (*Machine in automatic mode*)
		MasterInStandstill : BOOL; (*Master axis standing still (state Standstill OR Errorstop)*)
	END_VAR
	VAR_OUTPUT
		EStopMaster : BOOL; (*Emergency stop master axis*)
		ControlVoltage : BOOL; (*Connected to digital output for 24V control voltage *)
		Release : BOOL; (*Release for MC_Power function blocks*)
	END_VAR
	VAR
		State : emuSprMachine_PowerState;
		R_TRIG_SwitchOn : R_TRIG;
		TOF_ControlVoltage : TOF;
		EStopRequest : BOOL;
	END_VAR
END_FUNCTION_BLOCK

FUNCTION_BLOCK SPR_MachineMode (*Selects the machine mode*)
	VAR_INPUT
		AxesInStandstill : BOOL; (*all axes in standstill*)
		MasterInStandstill : BOOL; (*master axis in standstill*)
		TriggerAutoMode : BOOL; (*positive edge triggers a transition to auto mode if all axes are in standstill*)
		TriggerManualMode : BOOL; (*positive edge triggers a transition to manual mode if master is in standstill*)
	END_VAR
	VAR_OUTPUT
		ManualModeActive : BOOL;
		AutoModeActive : BOOL;
	END_VAR
	VAR
		MachineMode : USINT;
		R_TRIG_TriggerAutoMode : R_TRIG;
		R_TRIG_TriggerManualMode : R_TRIG;
	END_VAR
END_FUNCTION_BLOCK

FUNCTION_BLOCK SPR_BatchProduction (*Triggers a reduction of the master velocity and stop of master when the end of a batch is reached*)
	VAR_INPUT
		Enable : BOOL; (*enable batch production*)
		ActVelocity : REAL; (*actual master velocity [Master Units / s]*)
		Deceleration : REAL; (*master deceleration [Master Units / s²]*)
		ActProductCount : UDINT; (*actual product count*)
		SetProductCount : UDINT; (*target product count*)
		ProductLength : REAL; (*product length [Master Units]*)
		DistanceAtReducedVel : REAL; (*distance to be travelled with reduced velocity [Master Units]*)
	END_VAR
	VAR_OUTPUT
		BatchComplete : BOOL; (*target product count reached, batch complete*)
		ReduceVelocity : BOOL; (*end of batch almost reached, reduce velocity*)
	END_VAR
	VAR
		StoppingDistance : REAL; (*braking distance to reach standstill at actual velocity*)
		RemainingDistance : REAL; (*remaining distance in batch*)
		DeltaCount : DINT; (*SetProductCount - ActProductCount*)
		State : USINT;
	END_VAR
END_FUNCTION_BLOCK
```

#### SPR_MachinePower.st - Indicates status of machine control voltage
```iecst
(********************************************************************
 * COPYRIGHT -- Bernecker + Rainer
 ********************************************************************
 * Library: UserSpilke
 * File: SPR_MachinePower.st
 * Author: knausenbergl
 * Created: December 13, 2012
 ********************************************************************
 * Implementation of library UserSpilke
 ********************************************************************)

(*<$Description$> Indicates status of machine control voltage </$Description$>*)
FUNCTION_BLOCK SPR_MachinePower

	R_TRIG_SwitchOn.CLK	:= SwitchOn;
	R_TRIG_SwitchOn();

	EStopRequest	:= NOT SafetyOk OR SwitchOff;

	CASE State OF

		//**********	DRIVES DISABLED, CONTROL VOLTAGE OFF	**********
		SPR_MACH_PWR_DISABLED:
			TOF_ControlVoltage.IN	:= FALSE;
			Release					:= FALSE;
			EStopMaster				:= TRUE;

			IF (NOT EStopRequest AND R_TRIG_SwitchOn.Q) THEN
				//switch on control voltage
				TOF_ControlVoltage.IN	:= TRUE;
				Release					:= TRUE;
				EStopMaster				:= FALSE;
				State	:= SPR_MACH_PWR_ENABLED;
			END_IF;

		//**********	DRIVES ENABLED, CONTROL VOLTAGE ON		**********
		SPR_MACH_PWR_ENABLED:
			TOF_ControlVoltage.IN	:= TRUE;
			Release					:= TRUE;
			EStopMaster				:= FALSE;

			IF (EStopRequest) THEN
				//switch off control voltage (delayed)
				TOF_ControlVoltage.IN	:= FALSE;

				IF (AutoModeActive) THEN
					//stop master axis first if axes are running synchronized
					EStopMaster	:= TRUE;
					State		:= SPR_MACH_PWR_ESTOP_AUTO;
				ELSE
					//disable drives
					Release			:= FALSE;
					EStopMaster		:= TRUE;
					State			:= SPR_MACH_PWR_DELAY_24V_OFF;
				END_IF;
			END_IF;

		//**********	ESTOP REQUESTED, MASTER STOPPING		**********
		SPR_MACH_PWR_ESTOP_AUTO:
			TOF_ControlVoltage.IN	:= FALSE;
			Release					:= TRUE;
			EStopMaster				:= TRUE;

			IF (NOT TOF_ControlVoltage.Q) THEN
				//timer expired, control voltage switched off
				Release	:= FALSE;
				State	:= SPR_MACH_PWR_DISABLED;
			ELSIF (MasterInStandstill) THEN
				//disable drives
				Release	:= FALSE;
				State	:= SPR_MACH_PWR_DELAY_24V_OFF;
			END_IF;

		//**********	DELAYED CONTROL VOLTAGE SWITCH OFF		**********
		SPR_MACH_PWR_DELAY_24V_OFF:
			TOF_ControlVoltage.IN	:= FALSE;
			Release					:= FALSE;
			EStopMaster				:= TRUE;

			IF (NOT TOF_ControlVoltage.Q) THEN
				//control voltage is switched off, go back to initial state
				State	:= SPR_MACH_PWR_DISABLED;
			END_IF;

		//**********	ERROR		**********
		SPR_MACH_PWR_ERROR:
			TOF_ControlVoltage.IN	:= FALSE;
			Release					:= FALSE;
			EStopMaster				:= TRUE;

		ELSE
			TOF_ControlVoltage.IN	:= FALSE;
			Release					:= FALSE;
			EStopMaster				:= TRUE;
			State	:= SPR_MACH_PWR_ERROR;

	END_CASE;

	TOF_ControlVoltage.PT	:= SwitchOffDelay;
	TOF_ControlVoltage();
	ControlVoltage	:= TOF_ControlVoltage.Q;

END_FUNCTION_BLOCK
```

#### SPR_MachineMode.st - Selects the machine mode
```iecst
(********************************************************************
 * COPYRIGHT -- Bernecker + Rainer
 ********************************************************************
 * Library: SprMachine
 * File: SPR_MachineMode.st
 * Author: knausenbergl
 * Created: January 02, 2013
 ********************************************************************
 * Implementation of library SprMachine
 ********************************************************************)

(*<$Description$> Selects the machine mode </$Description$>*)
FUNCTION_BLOCK SPR_MachineMode

	R_TRIG_TriggerAutoMode.CLK	:= TriggerAutoMode;
	R_TRIG_TriggerAutoMode();

	R_TRIG_TriggerManualMode.CLK	:= TriggerManualMode;
	R_TRIG_TriggerManualMode();

	CASE MachineMode OF

		//MANUAL MODE
		0:
			IF (AxesInStandstill AND (R_TRIG_TriggerAutoMode.Q AND NOT R_TRIG_TriggerManualMode.Q) ) THEN
				MachineMode	:= 1;
			END_IF;

		//AUTO MODE
		1:
			IF (MasterInStandstill AND (R_TRIG_TriggerManualMode.Q AND NOT R_TRIG_TriggerAutoMode.Q) ) THEN
				MachineMode	:= 0;
			END_IF;

		//UNDEFINED, ERROR
		255:

		ELSE
			MachineMode	:= 255;

	END_CASE;

	ManualModeActive	:= (MachineMode = 0);
	AutoModeActive		:= (MachineMode = 1);

END_FUNCTION_BLOCK
```

#### SPR_BatchProduction.st - Triggers a reduction of the master velocity and stop of master when the end of a batch is reached
```iecst
(********************************************************************
 * COPYRIGHT -- Bernecker + Rainer
 ********************************************************************
 * Library: SprMachine
 * File: SPR_BatchProduction.st
 * Author: knausenbergl
 * Created: January 08, 2013
 ********************************************************************
 * Implementation of library SprMachine
 ********************************************************************)

(*<$Description$> Triggers a reduction of the master velocity and stop of master when the end of a batch is reached </$Description$>*)
FUNCTION_BLOCK SPR_BatchProduction

	DeltaCount			:= UDINT_TO_DINT(SetProductCount - ActProductCount);
	RemainingDistance	:= DINT_TO_REAL(DeltaCount) * ProductLength;

	//calculate stopping distance
	IF (Deceleration > 0.0) THEN
		StoppingDistance	:= 0.5 * ActVelocity**2 / Deceleration;
	ELSE
		StoppingDistance	:= 0.0;
	END_IF;

	//ANY STATE
	IF (NOT Enable) THEN
		ReduceVelocity	:= FALSE;
		BatchComplete	:= FALSE;
		State	:= 0;
	END_IF;

	CASE State OF
		//BATCH PRODUCTION DISABLED
		0:
			ReduceVelocity	:= FALSE;
			BatchComplete	:= FALSE;

			IF (Enable) THEN
				State	:= 1;
			END_IF;

		//BATCH PRODUCTION ACTIVE
		1:
			IF (RemainingDistance <= (StoppingDistance + DistanceAtReducedVel) ) THEN
				ReduceVelocity	:= TRUE;
				State			:= 2;
			END_IF;

		//BATCH COMPLETION AT REDUCED VELOCITY
		2:
			IF (DeltaCount <= 0) THEN
				ReduceVelocity	:= FALSE;
				BatchComplete	:= TRUE;
				State			:= 3;
			END_IF;

		//BATCH COMPLETE, WAITING FOR RESET
		3:

		//ERROR
		255:

		//STATE UNDEFINED
		ELSE
			State	:= 255;

	END_CASE;

END_FUNCTION_BLOCK
```

### Library Logical/Libraries/SprManual (IEC) - Axis handling for manual operation

#### SprManual.fun - Exported functions and function blocks
```iecst
(********************************************************************
 * COPYRIGHT -- Bernecker + Rainer
 ********************************************************************
 * Library: SprManual
 * File: SprManual.fun
 * Author: knausenbergl
 * Created: January 01, 2013
 ********************************************************************
 * Functions and function blocks of library SprManual
 ********************************************************************)

FUNCTION_BLOCK SPR_ManualMoveRelease (*Release manual movements*)
	VAR_INPUT
		ManualModeActive : BOOL; (*machine is in manual mode*)
		AxisPower : BOOL; (*axis is powered on*)
		AxisError : BOOL; (*FubError OR AxisError*)
		Reset : BOOL; (*reset output*)
	END_VAR
	VAR_OUTPUT
		Out : BOOL; (*give release for manual movements*)
	END_VAR
END_FUNCTION_BLOCK

FUNCTION_BLOCK SPR_ManualMove (*Start a manual movement*)
	VAR_INPUT
		In : BOOL; (*start command*)
		ManualMoveRelease : BOOL;
		AxisInStandstill : BOOL; (*axis in standstill state*)
	END_VAR
	VAR_OUTPUT
		Out : BOOL; (*starts movement (connected to FUB)*)
		Lock : BOOL; (*conditions to start a movement not met, output cannot be set*)
	END_VAR
	VAR
		R_TRIG_In : R_TRIG;
		RS_Out : RS;
	END_VAR
END_FUNCTION_BLOCK

FUNCTION_BLOCK SPR_ManualStop (*Triggers a stop movement*)
	VAR_INPUT
		In : BOOL; (*stop command*)
		ManualModeActive : BOOL; (*machine is in manual mode*)
		ManualMoveRelease : BOOL;
		AxisPower : BOOL; (*axis is powered on*)
	END_VAR
	VAR_OUTPUT
		Out : BOOL; (*stop movement (connected to FUB)*)
	END_VAR
	VAR
		R_TRIG_ManualMoveRelease : R_TRIG;
		F_TRIG_ManualMoveRelease : F_TRIG;
	END_VAR
END_FUNCTION_BLOCK
```

#### SPR_ManualMoveRelease.st - Release manual movements
```iecst
(********************************************************************
 * COPYRIGHT -- Bernecker + Rainer
 ********************************************************************
 * Library: SprManual
 * File: SPR_ManualRelease.st
 * Author: knausenbergl
 * Created: January 01, 2013
 ********************************************************************
 * Implementation of library SprManual
 ********************************************************************)

(*<$Description$> Release manual movements </$Description$>*)
FUNCTION_BLOCK SPR_ManualMoveRelease

	Out	:= ManualModeActive AND AxisPower AND NOT AxisError AND NOT Reset;

END_FUNCTION_BLOCK
```

#### SPR_ManualMove.st - Start a manual movement
```iecst
(********************************************************************
 * COPYRIGHT -- Bernecker + Rainer
 ********************************************************************
 * Library: SprManual
 * File: SPR_ManualMove.st
 * Author: knausenbergl
 * Created: January 01, 2013
 ********************************************************************
 * Implementation of library SprManual
 ********************************************************************)

(*<$Description$> Start a manual movement </$Description$>*)
FUNCTION_BLOCK SPR_ManualMove

	R_TRIG_In.CLK	:= In;
	R_TRIG_In();

	Lock	:= NOT( (AxisInStandstill OR Out) AND ManualMoveRelease);

	RS_Out.RESET1	:= NOT In OR NOT ManualMoveRelease;
	RS_Out.SET		:= R_TRIG_In.Q AND AxisInStandstill;
	RS_Out();
	Out	:= RS_Out.Q1;

END_FUNCTION_BLOCK
```

#### SPR_ManualStop.st - Triggers a stop movement
```iecst
(********************************************************************
 * COPYRIGHT -- Bernecker + Rainer
 ********************************************************************
 * Library: SprManual
 * File: SPR_ManualStop.st
 * Author: knausenbergl
 * Created: January 01, 2013
 ********************************************************************
 * Implementation of library SprManual
 ********************************************************************)

(*<$Description$> Triggers a stop movement </$Description$>*)
FUNCTION_BLOCK SPR_ManualStop

	R_TRIG_ManualMoveRelease.CLK	:= ManualMoveRelease;
	R_TRIG_ManualMoveRelease();

	F_TRIG_ManualMoveRelease.CLK	:= ManualMoveRelease;
	F_TRIG_ManualMoveRelease();

	Out	:= AxisPower AND ManualModeActive AND (In OR R_TRIG_ManualMoveRelease.Q OR F_TRIG_ManualMoveRelease.Q);

END_FUNCTION_BLOCK
```

### Library Logical/Libraries/SprSetup (IEC) - Axis handling for axis setup

#### SprSetup.fun - Exported functions and function blocks
```iecst
(********************************************************************
 * COPYRIGHT -- Bernecker + Rainer
 ********************************************************************
 * Library: SprSetup
 * File: SprSetup.fun
 * Author: knausenbergl
 * Created: January 15, 2013
 ********************************************************************
 * Functions and function blocks of library SprSetup
 ********************************************************************)

FUNCTION_BLOCK SPR_SetupRelease (*Give release for a setup operation*)
	VAR_INPUT
		AxisPower : BOOL; (*axis is powered on*)
		NetworkInit : BOOL; (*network initialized*)
		AxisError : BOOL; (*FubError OR AxisError*)
		Reset : BOOL; (*reset output*)
	END_VAR
	VAR_OUTPUT
		Out : BOOL; (*give release for setup operations (tuning, endcoder_if, ...)*)
	END_VAR
END_FUNCTION_BLOCK

FUNCTION_BLOCK SPR_Setup (*Start a setup operation*)
	VAR_INPUT
		In : BOOL;
		SetupRelease : BOOL;
		AxisDisabled : BOOL; (*axis in state disabled*)
	END_VAR
	VAR_OUTPUT
		Out : BOOL; (*triggers FUB*)
		Lock : BOOL; (*conditions to start setup operation not met, output cannot be set*)
	END_VAR
	VAR
		R_TRIG_In : R_TRIG;
		RS_Out : RS;
	END_VAR
END_FUNCTION_BLOCK
```

#### SPR_SetupRelease.st - Give release for a setup operation
```iecst
(********************************************************************
 * COPYRIGHT -- Bernecker + Rainer
 ********************************************************************
 * Library: SprSetup
 * File: SPR_SetupRelease.st
 * Author: knausenbergl
 * Created: January 15, 2013
 ********************************************************************
 * Implementation of library SprSetup
 ********************************************************************)

(*<$Description$> Give release for a setup operation </$Description$>*)
FUNCTION_BLOCK SPR_SetupRelease

	Out	:= NOT AxisPower AND NetworkInit AND NOT AxisError AND NOT Reset;

END_FUNCTION_BLOCK
```

#### SPR_Setup.st - Start a setup operation
```iecst
(********************************************************************
 * COPYRIGHT -- Bernecker + Rainer
 ********************************************************************
 * Library: SprSetup
 * File: SPR_Setup.st
 * Author: knausenbergl
 * Created: January 15, 2013
 ********************************************************************
 * Implementation of library SprSetup
 ********************************************************************)

(*<$Description$> Start a setup operation </$Description$>*)
FUNCTION_BLOCK SPR_Setup

	R_TRIG_In.CLK	:= In;
	R_TRIG_In();

	Lock	:= NOT( (AxisDisabled OR Out) AND SetupRelease);

	RS_Out.RESET1	:= NOT In OR NOT SetupRelease;
	RS_Out.SET		:= R_TRIG_In.Q AND AxisDisabled;
	RS_Out();
	Out	:= RS_Out.Q1;

END_FUNCTION_BLOCK
```

### Library Logical/Libraries/SprRegMa (IEC, version 1.00.0) - RegMark correction
Depends on: Acp10_MC, standard, SprGeneral

#### SprRegMa.typ - Exported data types
```iecst
(********************************************************************
 * COPYRIGHT -- Bernecker + Rainer
 ********************************************************************
 * Library: UserRegMa
 * File: UserRegMa.typ
 * Author: knausenbergl
 * Created: October 19, 2012
 ********************************************************************
 * Data types of library UserRegMa
 ********************************************************************)

TYPE
	emuSprRmState :
		(
		SPRRM_FIFO_DISABLED,
		SPRRM_FIFO_EMPTY,
		SPRRM_FIFO_EVALUATION_BUSY,
		SPRRM_FIFO_EVALUATION_DONE
		);
	SPR_RMCAPTURE_IS_TYP : 	STRUCT
		MC_BR_TouchProbe_0 : MC_BR_TouchProbe;
		SPR_RmCalcPosError_0 : SPR_RmCalcPosError;
		R_TRIG_Enable : R_TRIG;
		R_TRIG_SearchRM : R_TRIG;
		ProbeCounter_1 : UDINT;
	END_STRUCT;
END_TYPE
```

#### SprRegMa.fun - Exported functions and function blocks
```iecst
(********************************************************************
 * COPYRIGHT -- Bernecker + Rainer
 ********************************************************************
 * Library: UserRegMa
 * File: UserRegMa.fun
 * Author: knausenbergl
 * Created: October 19, 2012
 ********************************************************************
 * Functions and function blocks of library UserRegMa
 ********************************************************************)

FUNCTION_BLOCK SPR_RmCalcPosError (*Calculates a position error for registration mark control*)
	VAR_INPUT
		Enable : BOOL;
		RecordedValue : DINT; (*Recorded RegMark position, e.g. from a MC_BR_Touchprobe instance [Master Units]*)
		RecordedValueValid : BOOL;
		CutMasterPosition : DINT; (*Uncorrected next cut position [Master Units]*)
		DistanceToSensor : DINT; (*Distance between tool and sensor [Master Units]*)
		RegMarkPosition : DINT; (*RegMark offset relative to cut position [Master Units]*)
		ProductLength : DINT; (*Product length [Master Units]*)

	END_VAR
	VAR_OUTPUT
		PositionError : DINT; (*Difference between corrected and uncorrected cut position [Master Units]*)
		PositionErrorValid : BOOL; (*TRUE for 1 cycle if "PositionError" is within current product cycle*)
	END_VAR
	VAR
		State : emuSprRmState;
		SPR_Fifo_0 : SPR_Fifo;
		CorrectedCutPosition : DINT;
		PositionErrorTemp : DINT;
	END_VAR
END_FUNCTION_BLOCK

FUNCTION_BLOCK SPR_RmCapture (*Touchprobe with built-in FIFO for RegMark correction in cross-cutter applications*)
	VAR_INPUT
		Enable : BOOL;
		TriggerInput : MC_BR_TRIGGER_REF; (*Input that is used as event source*)
		Axis : UDINT; (*Axis reference of slave*)
		SearchRM : BOOL; (*Initiate search of new RM on positive edge*)
		CutMasterPosition : DINT; (*Uncorrected next cut position [Master Units]*)
		RegMarkPosition : DINT; (*RegMark offset relative to cut position [Master Units]*)
		WindowNegative : REAL; (*Range before the expected position in which the trigger signal may occur [Master Units]*)
		WindowPositive : REAL; (*Range after the expected position in which the trigger signal may occur [Master Units]*)
		ProductLength : REAL; (*Interval between two expected trigger positions [Master Units]*)
		DistanceToSensor : DINT; (*Distance between tool and sensor [Master Units]*)
	END_VAR
	VAR_OUTPUT
		RecordedValue : DINT; (*Most recent RM position [Master Units]*)
		ProbeCounter : UDINT; (*Number of valid trigger events. Reset by "SearchRM"*)
		MissedTriggers : UDINT; (*Number of invalid or missed trigger events. Reset by "SearchRM"*)
		CorrectionValue : DINT; (*Deviation between corrected and uncorrected cut position [Master Units]. Can be used as a relative distance for correction movements.*)
		CorrectionValid : BOOL; (*TRUE for 1 cycle if "CorrectionValue" is valid. Can be used to trigger correction movements.*)
		ActProductLength : REAL; (*Actual measured product length*)
		Active : BOOL; (*FB is enabled - waiting for a trigger event*)
		Busy : BOOL; (*FB is not yet finished*)
		Error : BOOL; (*Error occurred in FB*)
		ErrorID : UINT; (*Error number*)
	END_VAR
	VAR
		IS : SPR_RMCAPTURE_IS_TYP; (*internal data structure*)
	END_VAR
END_FUNCTION_BLOCK

FUNCTION_BLOCK SPR_RmPeriodicPosition (*Converts a DINT RegMark position into a periodic REAL RegMark position*)
	VAR_INPUT
		RecordedValue : DINT; (*Recorded RegMark position in DINT format [Master Units]*)
		MasterPeriodicPosition : REAL; (*Periodic master position in REAL format [Master Units]*)
		MasterPosition : DINT; (*Non-periodic master position in DINT format (from axis structure) [Master Units]*)
		MasterPeriod : DINT; (*Master axis modulo period [Master Units]*)
	END_VAR
	VAR_OUTPUT
		Out : REAL; (*Periodic RegMark position in REAL format [Master Units]*)
	END_VAR
	VAR
		MasterModuloOffset : DINT;
		RmModuloOffset : DINT;
		DeltaPeriods : DINT;
	END_VAR
END_FUNCTION_BLOCK
```

#### SPR_RmCalcPosError.st - Calculates a position error for registration mark control
```iecst
(********************************************************************
 * COPYRIGHT -- Bernecker + Rainer
 ********************************************************************
 * Library: UserRegMa
 * File: CalcPosError.st
 * Author: knausenbergl
 * Created: October 19, 2012
 ********************************************************************
 * Implementation of library UserRegMa
 ********************************************************************)
(*<$Description$> Calculates a position error for registration mark control </$Description$>*)
FUNCTION_BLOCK SPR_RmCalcPosError
	//save registration mark position in FIFO
	SPR_Fifo_0.InValue	:= RecordedValue;
	SPR_Fifo_0.Reset	:= NOT Enable;
	SPR_Fifo_0.Add		:= RecordedValueValid AND Enable;
	SPR_Fifo_0();

	//********************************	FIFO state-machine	**************************
	//Any state
	IF (NOT Enable) THEN
		State	:= SPRRM_FIFO_DISABLED;
	END_IF;

	CASE State OF
		//FIFO is disabled, waiting for Enable
		SPRRM_FIFO_DISABLED:
			PositionErrorValid	:= FALSE;
			PositionError		:= 0;

			IF (Enable) THEN
				State	:= SPRRM_FIFO_EMPTY;
			END_IF;

		//FIFO is enabled and empty
		SPRRM_FIFO_EMPTY:
			IF (SPR_Fifo_0.ActElements > 0) THEN
				State		:= SPRRM_FIFO_EVALUATION_BUSY;
			END_IF;

		//FIFO output value is under evaluation
		SPRRM_FIFO_EVALUATION_BUSY:
			CorrectedCutPosition	:= SPR_Fifo_0.OutValue + DistanceToSensor - RegMarkPosition;
			PositionErrorTemp		:= CorrectedCutPosition - CutMasterPosition;
			PositionError			:= PositionErrorTemp MOD ProductLength;

			IF (PositionErrorTemp > (- ProductLength / 2) ) THEN
				//wait until registration mark is within current product cycle
				IF (ABS(PositionErrorTemp) < (ProductLength / 2) ) THEN
					PositionErrorValid	:= TRUE;
					SPR_Fifo_0.Remove	:= TRUE;
					State				:= SPRRM_FIFO_EVALUATION_DONE;
				ELSIF (ABS(PositionErrorTemp) > (2 * DistanceToSensor) ) THEN
					//if position error is too large, it is assumed to be invalid
					SPR_Fifo_0.Remove	:= TRUE;
					State			:= SPRRM_FIFO_EVALUATION_DONE;
				END_IF;
			ELSE
				SPR_Fifo_0.Remove	:= TRUE;
				State				:= SPRRM_FIFO_EVALUATION_DONE;
			END_IF;

		//FIFO value has been evaluated, read next value
		SPRRM_FIFO_EVALUATION_DONE:
			SPR_Fifo_0.Remove			:= FALSE;
			PositionErrorValid		:= FALSE;

			IF (SPR_Fifo_0.ActElements > 0) THEN
				State		:= SPRRM_FIFO_EVALUATION_BUSY;
			ELSE
				State		:= SPRRM_FIFO_EMPTY;
			END_IF;

	END_CASE;

END_FUNCTION_BLOCK
```

#### SPR_RmCapture.st - Touchprobe with built-in FIFO for RegMark correction in cross-cutter applications
```iecst
(********************************************************************
 * COPYRIGHT -- Bernecker + Rainer
 ********************************************************************
 * Library: UserRegMa
 * File: CalcPosError.st
 * Author: knausenbergl
 * Created: October 19, 2012
 ********************************************************************
 * Implementation of library UserRegMa
 ********************************************************************)
(*<$Description$> Touchprobe with built-in FIFO for RegMark correction in cross-cutter applications </$Description$>*)
FUNCTION_BLOCK SPR_RmCapture

	IS.R_TRIG_Enable.CLK	:= Enable;
	IS.R_TRIG_Enable();

	IS.R_TRIG_SearchRM.CLK	:= SearchRM;
	IS.R_TRIG_SearchRM();

	//Enable positive edge
	IF (IS.R_TRIG_Enable.Q) THEN
		IS.MC_BR_TouchProbe_0.Axis				:= Axis;
		IS.MC_BR_TouchProbe_0.Period			:= ProductLength;
		IS.MC_BR_TouchProbe_0.PeriodChange		:= 0.0;
		IS.MC_BR_TouchProbe_0.ExpectedValue		:= 0.0;
		IS.MC_BR_TouchProbe_0.Mode				:= mcSHIFT_FROM_RESULT + mcUSE_FIRST_TRIGGER_POS;
		IS.MC_BR_TouchProbe_0.TriggerInput		:= TriggerInput;
		IS.MC_BR_TouchProbe_0.WindowNegative	:= WindowNegative;
		IS.MC_BR_TouchProbe_0.WindowPositive	:= WindowPositive;
		IS.SPR_RmCalcPosError_0.DistanceToSensor	:= DistanceToSensor;
		IS.SPR_RmCalcPosError_0.ProductLength		:= REAL_TO_DINT(ProductLength);

	//SearchRM positive edge
	ELSIF (Enable AND IS.R_TRIG_SearchRM.Q) THEN
		IS.MC_BR_TouchProbe_0.Axis				:= Axis;
		IS.MC_BR_TouchProbe_0.Period			:= ProductLength;
		IS.MC_BR_TouchProbe_0.PeriodChange		:= 0.0;
		IS.MC_BR_TouchProbe_0.ExpectedValue		:= 0.0;
		IS.MC_BR_TouchProbe_0.Mode				:= mcSHIFT_FROM_RESULT + mcUSE_FIRST_TRIGGER_POS;
		IS.MC_BR_TouchProbe_0.TriggerInput		:= TriggerInput;
		IS.MC_BR_TouchProbe_0.WindowNegative	:= WindowNegative;
		IS.MC_BR_TouchProbe_0.WindowPositive	:= WindowPositive;
		IS.SPR_RmCalcPosError_0.DistanceToSensor	:= DistanceToSensor;
		IS.SPR_RmCalcPosError_0.ProductLength		:= REAL_TO_DINT(ProductLength);
	END_IF;

	//disable TouchProbe on positive edge of "SearchRM" to re-initialize it
	IF (IS.R_TRIG_SearchRM.Q OR NOT Enable) THEN
		IS.MC_BR_TouchProbe_0.Enable	:= FALSE;
		IS.SPR_RmCalcPosError_0.Enable	:= FALSE;
	//wait until TouchProbe is inactive before restarting it
	ELSIF (Enable AND NOT IS.MC_BR_TouchProbe_0.Busy AND NOT IS.MC_BR_TouchProbe_0.Active) THEN
		IS.MC_BR_TouchProbe_0.Enable	:= TRUE;
		IS.SPR_RmCalcPosError_0.Enable	:= TRUE;
	END_IF;

	IS.MC_BR_TouchProbe_0();

	IS.SPR_RmCalcPosError_0.CutMasterPosition	:= CutMasterPosition;
	IS.SPR_RmCalcPosError_0.RecordedValue		:= IS.MC_BR_TouchProbe_0.RecordedValue;
	IS.SPR_RmCalcPosError_0.RecordedValueValid	:= IS.MC_BR_TouchProbe_0.Active AND (IS.MC_BR_TouchProbe_0.ProbeCounter <> IS.ProbeCounter_1);
	IS.SPR_RmCalcPosError_0.RegMarkPosition		:= RegMarkPosition;
	IS.SPR_RmCalcPosError_0.Enable				:= IS.MC_BR_TouchProbe_0.Busy;
	IS.SPR_RmCalcPosError_0();
	IS.ProbeCounter_1	:= IS.MC_BR_TouchProbe_0.ProbeCounter;

	//update FUB outputs
	RecordedValue		:= IS.MC_BR_TouchProbe_0.RecordedValue;
	ProbeCounter		:= IS.MC_BR_TouchProbe_0.ProbeCounter;
	MissedTriggers		:= IS.MC_BR_TouchProbe_0.MissedTriggers;
	CorrectionValue		:= IS.SPR_RmCalcPosError_0.PositionError;
	CorrectionValid		:= IS.SPR_RmCalcPosError_0.PositionErrorValid;
	Busy				:= Enable OR IS.MC_BR_TouchProbe_0.Busy;
	Active				:= IS.MC_BR_TouchProbe_0.Active;

	IF (IS.MC_BR_TouchProbe_0.Active) THEN
		ActProductLength	:= IS.MC_BR_TouchProbe_0.Period - IS.MC_BR_TouchProbe_0.DeltaExpectedValue;
	ELSE
		ActProductLength	:= 0.0;
	END_IF;

	IF (IS.MC_BR_TouchProbe_0.Enable) THEN
		Error	:= IS.MC_BR_TouchProbe_0.Error;
		ErrorID	:= IS.MC_BR_TouchProbe_0.ErrorID;
	ELSIF (NOT Enable) THEN
		Error	:= FALSE;
		ErrorID	:= FALSE;
	END_IF;

END_FUNCTION_BLOCK
```

#### SPR_RmPeriodicPosition.st - Converts a DINT RegMark position into a periodic REAL RegMark position
```iecst
(********************************************************************
 * COPYRIGHT -- Bernecker + Rainer
 ********************************************************************
 * Library: SprRegMa
 * File: SPR_RmPeriodicPosition.st
 * Author: knausenbergl
 * Created: January 25, 2013
 ********************************************************************
 * Implementation of library SprRegMa
 ********************************************************************)

(*<$Description$> Converts a DINT RegMark position into a periodic REAL RegMark position </$Description$>*)
FUNCTION_BLOCK SPR_RmPeriodicPosition
	IF (MasterPeriod > 0) THEN
		MasterModuloOffset	:= MasterPosition - REAL_TO_DINT(MasterPeriodicPosition);
		IF ( (RecordedValue - MasterModuloOffset) < 0) THEN
			DeltaPeriods	:= ( (RecordedValue - MasterModuloOffset) / MasterPeriod) - 1;
		ELSE
			DeltaPeriods	:= (RecordedValue - MasterModuloOffset) / MasterPeriod;
		END_IF;
		RmModuloOffset		:= MasterModuloOffset + (DeltaPeriods * MasterPeriod);
		Out					:= DINT_TO_REAL(RecordedValue - RmModuloOffset);
	ELSE
		Out	:= DINT_TO_REAL(RecordedValue);
	END_IF;
END_FUNCTION_BLOCK
```

### Library Logical/Libraries/SprGeneral (IEC) - Spilker general function blocks

#### SprGeneral.fun - Exported functions and function blocks
```iecst
(********************************************************************
 * COPYRIGHT -- Bernecker + Rainer
 ********************************************************************
 * Library: SprGeneral
 * File: SprGeneral.fun
 * Author: knausenbergl
 * Created: January 02, 2013
 ********************************************************************
 * Functions and function blocks of library SprGeneral
 ********************************************************************)

FUNCTION_BLOCK SPR_Mux (*Multiplexes pointers of any datatype*)
	VAR_INPUT
		Selector : USINT; (*Selects the channel*)
		pIn : ARRAY[0..15] OF UDINT; (*Addresses of input variables*)
	END_VAR
	VAR_OUTPUT
		Out_UDINT : UDINT; (*Output interpreted as UDINT*)
		Out_DINT : DINT; (*Output interpreted as DINT*)
		Out_REAL : REAL; (*Output interpreted as REAL*)
		Out_BOOL : BOOL;
		Out_USINT : USINT;
		Out_UINT : UINT;
		Out_INT : INT;
	END_VAR
	VAR
		C_Selector : USINT;
	END_VAR
END_FUNCTION_BLOCK

FUNCTION_BLOCK SPR_Fifo (*Implementation of a DINT Fifo*)
	VAR_INPUT
		Add : BOOL; (*add value to FIFO on positive edge*)
		Remove : BOOL; (*remove value from FIFO on positive edge*)
		InValue : DINT; (*input value for add command*)
		Reset : BOOL; (*reset FIFO on positive edge*)
	END_VAR
	VAR_OUTPUT
		Full : BOOL; (*FIFO is full*)
		ActElements : UINT; (*actual number of elements in FIFO*)
		OutValue : DINT; (*output value*)
	END_VAR
	VAR
		Add_1 : USINT; (*value in previous cycle*)
		Remove_1 : USINT; (*value in previous cycle*)
		Reset_1 : USINT; (*value in previous cycle*)
		RemoveIndex : USINT; (*remove index in value array*)
		AddIndex : USINT; (*add index in value array*)
		Value : ARRAY[0..255] OF DINT; (*value array*)
		MaxElements : UINT; (*maximum number of elements in FIFO*)
	END_VAR
END_FUNCTION_BLOCK
```

#### SPR_Mux.st - Multiplexes pointers of any datatype
```iecst
(********************************************************************
 * COPYRIGHT -- Bernecker + Rainer
 ********************************************************************
 * Library: SprGeneral
 * File: SPR_Mux.st
 * Author: knausenbergl
 * Created: January 02, 2013
 ********************************************************************
 * Implementation of library SprGeneral
 ********************************************************************)

(*<$Description$> Multiplexes pointers of any datatype </$Description$>*)
FUNCTION_BLOCK SPR_Mux

	C_Selector	:= LIMIT(0, Selector, (SIZEOF(pIn) / SIZEOF(pIn[0]) - 1) );

	IF (pIn[C_Selector] <> 0) THEN
		memcpy(ADR(Out_UDINT), pIn[C_Selector], SIZEOF(Out_UDINT) );
		memcpy(ADR(Out_DINT), pIn[C_Selector], SIZEOF(Out_DINT) );
		memcpy(ADR(Out_REAL), pIn[C_Selector], SIZEOF(Out_REAL) );
		memcpy(ADR(Out_BOOL), pIn[C_Selector], SIZEOF(Out_BOOL) );
		memcpy(ADR(Out_USINT), pIn[C_Selector], SIZEOF(Out_USINT) );
		memcpy(ADR(Out_INT), pIn[C_Selector], SIZEOF(Out_INT) );
		memcpy(ADR(Out_UINT), pIn[C_Selector], SIZEOF(Out_UINT) );
	END_IF;

END_FUNCTION_BLOCK
```

#### SPR_Fifo.st - Implementation of a DINT Fifo
```iecst
(********************************************************************
 * COPYRIGHT -- Bernecker + Rainer
 ********************************************************************
 * Library: Fifo
 * File: Fifo.st
 * Author: knausenbergl
 * Created: October 19, 2012
 ********************************************************************
 * Implementation of library Fifo
 ********************************************************************)

(*<$Description$> Implementation of a DINT Fifo </$Description$>*)
FUNCTION_BLOCK SPR_Fifo
	MaxElements	:= SIZEOF(Value)/SIZEOF(Value[0]);

	//reset FIFO
	IF (Reset > Reset_1) THEN
		memset(ADR(Value), 0, SIZEOF(Value) );
		AddIndex	:= 0;
		RemoveIndex	:= 0;
		ActElements	:= 0;
	END_IF;
	Reset_1	:= Reset;

	//remove value from FIFO
	IF (Remove > Remove_1) THEN
		IF (ActElements >= 1) THEN
			Value[RemoveIndex]	:= 0;
			RemoveIndex			:= UINT_TO_USINT( (RemoveIndex + 1) MOD MaxElements);
			ActElements			:= ActElements - 1;
		END_IF;
	END_IF;
	Remove_1	:= Remove;

	//add value to FIFO
	IF (Add > Add_1) THEN
		IF (ActElements < MaxElements) THEN
			Value[AddIndex]		:= InValue;
			AddIndex			:= UINT_TO_USINT( (AddIndex + 1) MOD MaxElements);
			ActElements			:= ActElements + 1;
		ELSE
		END_IF;
	END_IF;
	Add_1	:= Add;

	OutValue	:= Value[RemoveIndex];
	Full		:= (ActElements >= MaxElements);

END_FUNCTION_BLOCK
```

### Data object Logical/acp10etxde (Ett)

- acp10etxde.ett (not shown)

### Package Logical/AxisObj - Paket

### Data object Logical/AxisObj/gunwfeedi (Ax)
